# B&R Automation Studio project ComauRacer3demo
Automation Studio 4.9.2.46; technology packages: mapp 5.14.1, mappCockpit 5.14.0, mappMotion 5.14.2, mappView 5.14.2

## Configuration Racer3_demo

CPU 5APC2100.BY44-000, AutomationRuntime C4.83, Build 4.1.2, Vc V4.72.2

### Task classes (Cpu.sw)
```
Cyclic#4:
  Control <- Racer3.Control.prg
Libraries: MpRobotics, McAxGroup, MpBase, McBase, CoTrace, AsZip, FileIO, runtime, MpAlarmX, astime, MpAudit, MpRecipe, sys_lib, MpServer, MpUserX
```

### AxesGrpR3.axesgroup - 5APC2100_BY44_000/mappMotion/ComauRacer3/AxesGrpR3.axesgroup
```
Element gAxesGroup (Type=axesgroup)
  Type = PathGenAxesGroup
    ProcessingTaskClass = 1
    License = 1
    PhysicalAxes:
      JointAxes:
        JointAxis[1]:
          Name = Q1
          AxisRef = gAxisQ1
        JointAxis[2]:
          Name = Q2
          AxisRef = gAxisQ2
        JointAxis[3]:
          Name = Q3
          AxisRef = gAxisQ3
        JointAxis[4]:
          Name = Q4
          AxisRef = gAxisQ4
        JointAxis[5]:
          Name = Q5
          AxisRef = gAxisQ5
        JointAxis[6]:
          Name = Q6
          AxisRef = gAxisQ6
    MechanicalSystem:
      MechSysRef = MechSysRacer3
    BasicSettings:
      ModalDataBehaviour = ResetToDefault
      GeometryPlanning:
        TCPResolution:
          LengthResolution = 0.001
          AngleResolution = 0.001
        RoundingMode = Standard
        MaxCornerDeviation = 0.0
        MaxTangentialTransitionDeviation = 0.05
        MaxRadiusDeviation = 0.001
        WorkingPlane = XY
      TrajectoryPlanning = Basic
        LimitCheckResolution = UserDefinedTime
          Time = 0.005
        BufferTime = UserDefinedTime
          Time = 0.050
    AxesGroupFeatures:
      FeatureRef[1] = FeatureProgramsRacer3
      FeatureRef[2] = FeatureFeedForwardRacer3
      FeatureRef[3] = FeatureJoggingRacer3
  Alarms = None
```

### MotionConf.mappmotioncfg - 5APC2100_BY44_000/mappMotion/MotionConf.mappmotioncfg
```
Element MappMotionConfiguration (Type=mappmotioncfg)
```

## Configuration Racer3_working

CPU 5APC2100.BY44-000, AutomationRuntime C4.83, Build 4.1.2, Vc V4.72.2

### Task classes (Cpu.sw)
```
Cyclic#1 (cycle 2000 us, tolerance 0 us):
  Control <- Racer3.Control.prg
Cyclic#4:
  Auditing <- Auditing.prg
  Alarm <- Alarm.prg
  FileManage <- FileManager.prg
DataObjects: McAcpSys
Binaries: TCLang, McAcpDrv, McAcpSim, mvLoader, arflatprv, udbdef, TCData, mCoWebSc, McMechSys, FWRules, arcoal, arsvcreg, McPathXT, Settings, iomap, AxesR3, Role, ashwac, Hierarchy, AxGrpFtrR3, asfw, sysconf, MechSysR3, arconfig, AxesGrpR3, TC, ashwd, User, Config, Config_1, FileMngMap, Workspace, FileMngUI, ConfigF, ConfigAlmH, ConfigAdt, ConfigAlm, Config_4, Config_3, Config_2
Libraries: operator, runtime, astime, AsIecCon, MpRobotics, McAxGroup, MpBase, McBase, CoTrace, AsZip, FileIO, sys_lib, McAcpAx, McAxis, RacerLib, MpAxis, McAcpPar, McPathGen, McProgInt, MpAudit, MpServer, MpAlarmX, MpFile, AsBrStr, arssl, powerlnk, asarprof, asarlog, asio, asmem, dataobj, asepl, brsystem, aruser, MpUserX, MpFile, asbrstr, asusb
```

### Hardware
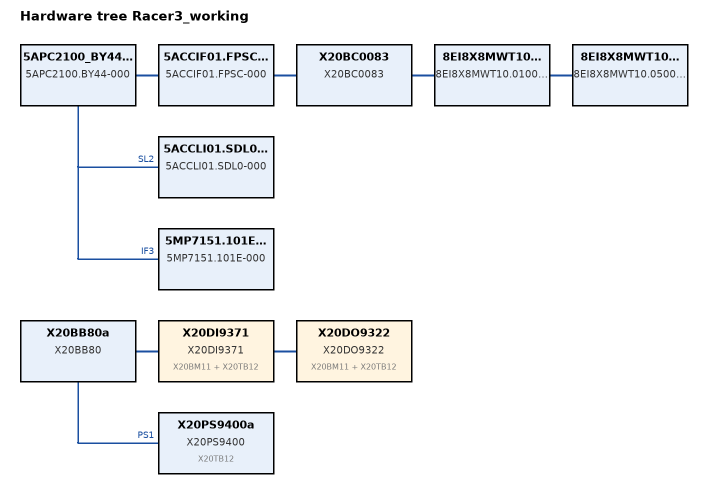
```
5ACCIF01.FPSC-000 : 5ACCIF01.FPSC-000 v1.9.0.3  [SL -> 5APC2100_BY44_000.SL1]
  Connector IF1:
    Channel1
    ChannelID1 = McAcpBroadcast
    ChannelType1 = OCTET[96]
5ACCLI01.SDL0-000 : 5ACCLI01.SDL0-000 v2.0.0.0  [SL -> 5APC2100_BY44_000.SL2]
5APC2100_BY44_000 : 5APC2100.BY44-000 v2.1.0.0
  Connector IF3:
    AssignedOperatingSystem = ARemb
    ActivateDevice = 1
    Mode = Manual
    InternetAddress = 192.168.0.100
    SubnetMask = 255.255.255.0
    ActivateSnmp = 2
  Connector IF4:
    AssignedOperatingSystem = ARemb
    ActivateDevice = 1
    Mode = Manual
    InternetAddress = 192.168.1.100
    SubnetMask = 255.255.255.0
    ActivateSnmp = 2
  Connector IF5:
    AssignedOperatingSystem = ARemb
  Connector IF6:
    AssignedOperatingSystem = ARemb
  ConfigurationID = ComauRacer3demo_czysty_racer3
  UserPartitionSize = 128
  Simulation = 1
  RemMemDevice = PCI.1.PPC21xx.SRAM
  RemMemSize = 2048
  PermanentPvSize = 768
  TimerDeviceType = EPLX2X
  TimerDevice = 5ACCIF01.FPSC-000.IF1
  TaskClassIdleTime = 2000
  Cyclic1Duration = 2000
  Cyclic1Tolerance = 0
  Cyclic1Output = 1
  FileDevice1
  FileDeviceName1 = CNC_PrgDir
  FileDevicePath1 = F:\CNC_PrgDir  // For HW config use D:\CNC_PrgDir\
  FileDevice2
  FileDeviceName2 = AUDIT
  FileDevicePath2 = F:\Audit
  FileDevice3
  FileDeviceName3 = UserPart
  FileDevicePath3 = F:\UserPart\  // For HW config use F:\
  FileDevice4
  FileDeviceName4 = RECIPE
  FileDevicePath4 = F:\Recipe
  TimeZone = 160
  ActivateDaylightSavingTime = 1
  FtpUser1
  FtpUsername1 = Admin
  FtpUserPassword1 = dPVRvIP+UG4zebJ0O0hf643aLF5yFibVmkrUfiZ9rkg=
  FtpUserSalt1 = Grtq2ClC
  FTPAccessRight1 = 0
  ActivateOpcUa = 1
  OpcUaActivateAuditEvents = 1
  OpcUa_Security_AdminRole = Everyone
  OpcUaInformationModels_PV_Version = 1
5MP7151.101E-000 : 5MP7151.101E-000 v1.1.0.0  [ETH1 -> 5APC2100_BY44_000.IF3 [Cable Type=PowerlinkCable, Length=10, Version=1.0.0.3]]
  Terminal = true
  VncKeyMappingFile = VC\5MP7151.101E-000.dis
  VncPortNumber = 5901
8EI8X8MWT10.0100-1 : 8EI8X8MWT10.0100-1 v2.3.0.3  [PLK1 -> X20BC0083.PLK2 (NodeNumber=4) [Cable Type=PowerlinkCable, Length=10, Version=1.0.0.3]; PLK2 -> 8EI8X8MWT10.0500-1.PLK1 (NodeNumber=4) [Cable Type=PowerlinkCable, Length=10, Version=1.0.0.3]]
  DriveConfiguration/Module:
    McAcoposTypeID = AcoposP3TConfig
    ActivateACOPOSSimulationOnPLC = 0
  DriveConfiguration/Encoder/EncoderX41:
    InterfaceType = EnDat
  DriveConfiguration/Encoder/EncoderX42:
    InterfaceType = EnDat
  DriveConfiguration/Encoder/EncoderX43:
    InterfaceType = EnDat
  DriveConfiguration/Channel[1]/RealAxis:
    AxisReference = gAxisQ1
  DriveConfiguration/Channel[1]/RealAxis/MechanicalElements/Gearbox:
    InputIsReadOnly = 1
    Input = 81818
    OutputIsReadOnly = 1
    Output = 1000
  DriveConfiguration/Channel[1]/RealAxis/MechanicalElements/RotaryToLinearTransformation:
    ReferenceDistanceIsReadOnly = 1
    ReferenceDistance = 360
  DriveConfiguration/Channel[1]/RealAxis/Controller:
    ModeIsReadOnly = 1
    Mode = PositionControllerWithTorqueFeedForward
  DriveConfiguration/Channel[1]/RealAxis/Controller/Mode/Position:
    ProportionalGainIsReadOnly = 1
    ProportionalGain = 75.0
    IntegrationTimeIsReadOnly = 1
    IntegrationTime = 0.0
    TotalDelayTime = 0.0004
  DriveConfiguration/Channel[1]/RealAxis/Controller/Mode/Speed:
    ProportionalGainIsReadOnly = 1
    ProportionalGain = 2.0
    IntegrationTimeIsReadOnly = 1
    IntegrationTime = 0.0
    FilterTimeIsReadOnly = 1
    FilterTime = 0.0008
  DriveConfiguration/Channel[1]/RealAxis/Controller/Mode:
    FeedForwardIsReadOnly = 1
    FeedForward = CyclicValueFromAxesGroup
  DriveConfiguration/Channel[1]/RealAxis/Controller/Mode/LoopFilters:
    LoopFilter1 = NotUsed
    LoopFilter2 = NotUsed
    LoopFilter3 = NotUsed
  DriveConfiguration/Channel[1]/RealAxis/Homing:
    Mode = RestorePosition
    RestorePositionVariable = ::gRacer3HomeRestorePos[0]
  DriveConfiguration/Channel[1]/RealAxis/StopReaction:
    Quickstop = DecelerationLimit
    DriveError = DecelerationLimit
  DriveConfiguration/Channel[1]/RealAxis/MovementErrorLimits:
    PositionError = 1.0
    VelocityErrorMonitoring = Automatic1
  DriveConfiguration/Channel[1]/RealAxis:
    JerkFilter = Used
  DriveConfiguration/Channel[1]/RealAxis/JerkFilter:
    JerkTime = 0.01
  DriveConfiguration/Channel[1]/RealAxis/DigitalInputs/HomingSwitch:
    Source = NotUsed
    Level = High
  DriveConfiguration/Channel[1]/RealAxis/DigitalInputs/PositiveLimitSwitch:
    Source = NotUsed
    Level = High
  DriveConfiguration/Channel[1]/RealAxis/DigitalInputs/NegativeLimitSwitch:
    Source = NotUsed
    Level = High
  DriveConfiguration/Channel[1]/RealAxis/DigitalInputs/Trigger1:
    Source = X8Trigger1
    Level = High
  DriveConfiguration/Channel[1]/RealAxis/DigitalInputs/Trigger2:
    Source = X8Trigger2
    Level = High
  DriveConfiguration/Channel[1]/RealAxis/DigitalInputs/Quickstop:
    Input = Trigger2
  DriveConfiguration/Channel[1]/RealAxis/Simulation:
    SimulationModeOnPLC = SetValueGeneration
    SimulationModeOnACOPOS = NotUsed
  DriveConfiguration/Channel[2]/RealAxis:
    AxisReference = gAxisQ3
  DriveConfiguration/Channel[2]/RealAxis/MechanicalElements/Gearbox:
    InputIsReadOnly = 1
    Input = 72
    OutputIsReadOnly = 1
    Output = 1
  DriveConfiguration/Channel[2]/RealAxis/MechanicalElements/RotaryToLinearTransformation:
    ReferenceDistanceIsReadOnly = 1
    ReferenceDistance = 360
  DriveConfiguration/Channel[2]/RealAxis/Controller:
    ModeIsReadOnly = 1
    Mode = PositionControllerWithTorqueFeedForward
  DriveConfiguration/Channel[2]/RealAxis/Controller/Mode/Position:
    ProportionalGainIsReadOnly = 1
    ProportionalGain = 50.0
    IntegrationTimeIsReadOnly = 1
    IntegrationTime = 0.0
    TotalDelayTime = 0.0004
  DriveConfiguration/Channel[2]/RealAxis/Controller/Mode/Speed:
    ProportionalGainIsReadOnly = 1
    ProportionalGain = 1.5
    IntegrationTimeIsReadOnly = 1
    IntegrationTime = 0.0
    FilterTimeIsReadOnly = 1
    FilterTime = 0.0008
  DriveConfiguration/Channel[2]/RealAxis/Controller/Mode:
    FeedForwardIsReadOnly = 1
    FeedForward = CyclicValueFromAxesGroup
  DriveConfiguration/Channel[2]/RealAxis/Controller/Mode/LoopFilters:
    LoopFilter1 = NotUsed
    LoopFilter2 = NotUsed
    LoopFilter3 = NotUsed
  DriveConfiguration/Channel[2]/RealAxis/Homing:
    Mode = RestorePosition
    RestorePositionVariable = ::gRacer3HomeRestorePos[2]
  DriveConfiguration/Channel[2]/RealAxis/StopReaction:
    Quickstop = DecelerationLimit
    DriveError = DecelerationLimit
  DriveConfiguration/Channel[2]/RealAxis/MovementErrorLimits:
    PositionError = 1.0
    VelocityErrorMonitoring = Automatic1
  DriveConfiguration/Channel[2]/RealAxis:
    JerkFilter = Used
  DriveConfiguration/Channel[2]/RealAxis/JerkFilter:
    JerkTime = 0.01
  DriveConfiguration/Channel[2]/RealAxis/DigitalInputs/HomingSwitch:
    Source = NotUsed
    Level = High
  DriveConfiguration/Channel[2]/RealAxis/DigitalInputs/PositiveLimitSwitch:
    Source = NotUsed
    Level = High
  DriveConfiguration/Channel[2]/RealAxis/DigitalInputs/NegativeLimitSwitch:
    Source = NotUsed
    Level = High
  DriveConfiguration/Channel[2]/RealAxis/DigitalInputs/Trigger1:
    Source = X8Trigger1
    Level = High
  DriveConfiguration/Channel[2]/RealAxis/DigitalInputs/Trigger2:
    Source = X8Trigger2
    Level = High
  DriveConfiguration/Channel[2]/RealAxis/DigitalInputs/Quickstop:
    Input = Trigger2
  DriveConfiguration/Channel[2]/RealAxis/Simulation:
    SimulationModeOnPLC = SetValueGeneration
    SimulationModeOnACOPOS = NotUsed
  DriveConfiguration/Channel[3]/RealAxis:
    AxisReference = gAxisQ5
  DriveConfiguration/Channel[3]/RealAxis/MechanicalElements/Gearbox:
    InputIsReadOnly = 1
    Input = 612
    OutputIsReadOnly = 1
    Output = 10
  DriveConfiguration/Channel[3]/RealAxis/MechanicalElements/RotaryToLinearTransformation:
    ReferenceDistanceIsReadOnly = 1
    ReferenceDistance = 360
  DriveConfiguration/Channel[3]/RealAxis/Controller:
    ModeIsReadOnly = 1
    Mode = PositionControllerWithTorqueFeedForward
  DriveConfiguration/Channel[3]/RealAxis/Controller/Mode/Position:
    ProportionalGainIsReadOnly = 1
    ProportionalGain = 200.0
    IntegrationTimeIsReadOnly = 1
    IntegrationTime = 0.0
    TotalDelayTime = 0.0004
  DriveConfiguration/Channel[3]/RealAxis/Controller/Mode/Speed:
    ProportionalGainIsReadOnly = 1
    ProportionalGain = 1.5
    IntegrationTimeIsReadOnly = 1
    IntegrationTime = 0.0
    FilterTimeIsReadOnly = 1
    FilterTime = 0.0008
  DriveConfiguration/Channel[3]/RealAxis/Controller/Mode:
    FeedForwardIsReadOnly = 1
    FeedForward = CyclicValueFromAxesGroup
  DriveConfiguration/Channel[3]/RealAxis/Controller/Mode/LoopFilters:
    LoopFilter1 = NotUsed
    LoopFilter2 = NotUsed
    LoopFilter3 = NotUsed
  DriveConfiguration/Channel[3]/RealAxis/Homing:
    Mode = RestorePosition
    RestorePositionVariable = ::gRacer3HomeRestorePos[4]
  DriveConfiguration/Channel[3]/RealAxis/StopReaction:
    Quickstop = DecelerationLimit
    DriveError = DecelerationLimit
  DriveConfiguration/Channel[3]/RealAxis/MovementErrorLimits:
    PositionError = 1.0
    VelocityErrorMonitoring = Automatic1
  DriveConfiguration/Channel[3]/RealAxis:
    JerkFilter = Used
  DriveConfiguration/Channel[3]/RealAxis/JerkFilter:
    JerkTime = 0.01
  DriveConfiguration/Channel[3]/RealAxis/DigitalInputs/HomingSwitch:
    Source = NotUsed
    Level = High
  DriveConfiguration/Channel[3]/RealAxis/DigitalInputs/PositiveLimitSwitch:
    Source = NotUsed
    Level = High
  DriveConfiguration/Channel[3]/RealAxis/DigitalInputs/NegativeLimitSwitch:
    Source = NotUsed
    Level = High
  DriveConfiguration/Channel[3]/RealAxis/DigitalInputs/Trigger1:
    Source = X8Trigger1
    Level = High
  DriveConfiguration/Channel[3]/RealAxis/DigitalInputs/Trigger2:
    Source = X8Trigger2
    Level = High
  DriveConfiguration/Channel[3]/RealAxis/DigitalInputs/Quickstop:
    Input = Trigger2
  DriveConfiguration/Channel[3]/RealAxis/Simulation:
    SimulationModeOnPLC = SetValueGeneration
    SimulationModeOnACOPOS = NotUsed
8EI8X8MWT10.0500-1 : 8EI8X8MWT10.0500-1 v2.3.0.3  [PLK1 -> 8EI8X8MWT10.0100-1.PLK2 (NodeNumber=5) [Cable Type=PowerlinkCable, Length=10, Version=1.0.0.3]]
  DriveConfiguration/Module:
    McAcoposTypeID = AcoposP3TConfig
    ActivateACOPOSSimulationOnPLC = 0
  DriveConfiguration/Encoder/EncoderX41:
    InterfaceType = EnDat
  DriveConfiguration/Encoder/EncoderX42:
    InterfaceType = EnDat
  DriveConfiguration/Encoder/EncoderX43:
    InterfaceType = EnDat
  DriveConfiguration/Channel[1]/RealAxis:
    AxisReference = gAxisQ2
  DriveConfiguration/Channel[1]/RealAxis/MechanicalElements/Gearbox:
    InputIsReadOnly = 1
    Input = 80
    OutputIsReadOnly = 1
    Output = 1
  DriveConfiguration/Channel[1]/RealAxis/MechanicalElements/RotaryToLinearTransformation:
    ReferenceDistanceIsReadOnly = 1
    ReferenceDistance = 360
  DriveConfiguration/Channel[1]/RealAxis/Controller:
    ModeIsReadOnly = 1
    Mode = PositionControllerWithTorqueFeedForward
  DriveConfiguration/Channel[1]/RealAxis/Controller/Mode/Position:
    ProportionalGainIsReadOnly = 1
    ProportionalGain = 50.0
    IntegrationTimeIsReadOnly = 1
    IntegrationTime = 0.0
    TotalDelayTime = 0.0004
  DriveConfiguration/Channel[1]/RealAxis/Controller/Mode/Speed:
    ProportionalGainIsReadOnly = 1
    ProportionalGain = 2.0
    IntegrationTimeIsReadOnly = 1
    IntegrationTime = 0.0
    FilterTimeIsReadOnly = 1
    FilterTime = 0.0008
  DriveConfiguration/Channel[1]/RealAxis/Controller/Mode:
    FeedForwardIsReadOnly = 1
    FeedForward = CyclicValueFromAxesGroup
  DriveConfiguration/Channel[1]/RealAxis/Controller/Mode/LoopFilters:
    LoopFilter1 = NotUsed
    LoopFilter2 = NotUsed
    LoopFilter3 = NotUsed
  DriveConfiguration/Channel[1]/RealAxis/Homing:
    Mode = RestorePosition
    RestorePositionVariable = ::gRacer3HomeRestorePos[1]
  DriveConfiguration/Channel[1]/RealAxis/StopReaction:
    Quickstop = DecelerationLimit
    DriveError = DecelerationLimit
  DriveConfiguration/Channel[1]/RealAxis/MovementErrorLimits:
    PositionError = 1.0
    VelocityErrorMonitoring = Automatic1
  DriveConfiguration/Channel[1]/RealAxis:
    JerkFilter = Used
  DriveConfiguration/Channel[1]/RealAxis/JerkFilter:
    JerkTime = 0.01
  DriveConfiguration/Channel[1]/RealAxis/DigitalInputs/HomingSwitch:
    Source = NotUsed
    Level = High
  DriveConfiguration/Channel[1]/RealAxis/DigitalInputs/PositiveLimitSwitch:
    Source = NotUsed
    Level = High
  DriveConfiguration/Channel[1]/RealAxis/DigitalInputs/NegativeLimitSwitch:
    Source = NotUsed
    Level = High
  DriveConfiguration/Channel[1]/RealAxis/DigitalInputs/Trigger1:
    Source = X8Trigger1
    Level = High
  DriveConfiguration/Channel[1]/RealAxis/DigitalInputs/Trigger2:
    Source = X8Trigger2
    Level = High
  DriveConfiguration/Channel[1]/RealAxis/DigitalInputs/Quickstop:
    Input = Trigger2
  DriveConfiguration/Channel[1]/RealAxis/Simulation:
    SimulationModeOnPLC = SetValueGeneration
    SimulationModeOnACOPOS = NotUsed
  DriveConfiguration/Channel[2]/RealAxis:
    AxisReference = gAxisQ4
  DriveConfiguration/Channel[2]/RealAxis/MechanicalElements/Gearbox:
    InputIsReadOnly = 1
    Input = 612
    OutputIsReadOnly = 1
    Output = 10
  DriveConfiguration/Channel[2]/RealAxis/MechanicalElements/RotaryToLinearTransformation:
    ReferenceDistanceIsReadOnly = 1
    ReferenceDistance = 360
  DriveConfiguration/Channel[2]/RealAxis/Controller:
    ModeIsReadOnly = 1
    Mode = PositionControllerWithTorqueFeedForward
  DriveConfiguration/Channel[2]/RealAxis/Controller/Mode/Position:
    ProportionalGainIsReadOnly = 1
    ProportionalGain = 100.0
    IntegrationTimeIsReadOnly = 1
    IntegrationTime = 0.0
    TotalDelayTime = 0.0004
  DriveConfiguration/Channel[2]/RealAxis/Controller/Mode/Speed:
    ProportionalGainIsReadOnly = 1
    ProportionalGain = 2.0
    IntegrationTimeIsReadOnly = 1
    IntegrationTime = 0.0
    FilterTimeIsReadOnly = 1
    FilterTime = 0.0008
  DriveConfiguration/Channel[2]/RealAxis/Controller/Mode:
    FeedForwardIsReadOnly = 1
    FeedForward = CyclicValueFromAxesGroup
  DriveConfiguration/Channel[2]/RealAxis/Controller/Mode/LoopFilters:
    LoopFilter1 = NotUsed
    LoopFilter2 = NotUsed
    LoopFilter3 = NotUsed
  DriveConfiguration/Channel[2]/RealAxis/Homing:
    Mode = RestorePosition
    RestorePositionVariable = ::gRacer3HomeRestorePos[3]
  DriveConfiguration/Channel[2]/RealAxis/StopReaction:
    Quickstop = DecelerationLimit
    DriveError = DecelerationLimit
  DriveConfiguration/Channel[2]/RealAxis/MovementErrorLimits:
    PositionError = 1.0
    VelocityErrorMonitoring = Automatic1
  DriveConfiguration/Channel[2]/RealAxis:
    JerkFilter = Used
  DriveConfiguration/Channel[2]/RealAxis/JerkFilter:
    JerkTime = 0.01
  DriveConfiguration/Channel[2]/RealAxis/DigitalInputs/HomingSwitch:
    Source = NotUsed
    Level = High
  DriveConfiguration/Channel[2]/RealAxis/DigitalInputs/PositiveLimitSwitch:
    Source = NotUsed
    Level = High
  DriveConfiguration/Channel[2]/RealAxis/DigitalInputs/NegativeLimitSwitch:
    Source = NotUsed
    Level = High
  DriveConfiguration/Channel[2]/RealAxis/DigitalInputs/Trigger1:
    Source = X8Trigger1
    Level = High
  DriveConfiguration/Channel[2]/RealAxis/DigitalInputs/Trigger2:
    Source = X8Trigger2
    Level = High
  DriveConfiguration/Channel[2]/RealAxis/DigitalInputs/Quickstop:
    Input = Trigger2
  DriveConfiguration/Channel[2]/RealAxis/Simulation:
    SimulationModeOnPLC = SetValueGeneration
    SimulationModeOnACOPOS = NotUsed
  DriveConfiguration/Channel[3]/RealAxis:
    AxisReference = gAxisQ6
  DriveConfiguration/Channel[3]/RealAxis/MechanicalElements/Gearbox:
    InputIsReadOnly = 1
    Input = 40
    OutputIsReadOnly = 1
    Output = 1
  DriveConfiguration/Channel[3]/RealAxis/MechanicalElements/RotaryToLinearTransformation:
    ReferenceDistanceIsReadOnly = 1
    ReferenceDistance = 360
  DriveConfiguration/Channel[3]/RealAxis/Controller:
    ModeIsReadOnly = 1
    Mode = PositionControllerWithTorqueFeedForward
  DriveConfiguration/Channel[3]/RealAxis/Controller/Mode/Position:
    ProportionalGainIsReadOnly = 1
    ProportionalGain = 200.0
    IntegrationTimeIsReadOnly = 1
    IntegrationTime = 0.0
    TotalDelayTime = 0.0004
  DriveConfiguration/Channel[3]/RealAxis/Controller/Mode/Speed:
    ProportionalGainIsReadOnly = 1
    ProportionalGain = 1.5
    IntegrationTimeIsReadOnly = 1
    IntegrationTime = 0.0
    FilterTimeIsReadOnly = 1
    FilterTime = 0.0008
  DriveConfiguration/Channel[3]/RealAxis/Controller/Mode:
    FeedForwardIsReadOnly = 1
    FeedForward = CyclicValueFromAxesGroup
  DriveConfiguration/Channel[3]/RealAxis/Controller/Mode/LoopFilters:
    LoopFilter1 = NotUsed
    LoopFilter2 = NotUsed
    LoopFilter3 = NotUsed
  DriveConfiguration/Channel[3]/RealAxis/Homing:
    Mode = RestorePosition
    RestorePositionVariable = ::gRacer3HomeRestorePos[5]
  DriveConfiguration/Channel[3]/RealAxis/StopReaction:
    Quickstop = DecelerationLimit
    DriveError = DecelerationLimit
  DriveConfiguration/Channel[3]/RealAxis/MovementErrorLimits:
    PositionError = 1.0
    VelocityErrorMonitoring = Automatic1
  DriveConfiguration/Channel[3]/RealAxis:
    JerkFilter = Used
  DriveConfiguration/Channel[3]/RealAxis/JerkFilter:
    JerkTime = 0.01
  DriveConfiguration/Channel[3]/RealAxis/DigitalInputs/HomingSwitch:
    Source = NotUsed
    Level = High
  DriveConfiguration/Channel[3]/RealAxis/DigitalInputs/PositiveLimitSwitch:
    Source = NotUsed
    Level = High
  DriveConfiguration/Channel[3]/RealAxis/DigitalInputs/NegativeLimitSwitch:
    Source = NotUsed
    Level = High
  DriveConfiguration/Channel[3]/RealAxis/DigitalInputs/Trigger1:
    Source = X8Trigger1
    Level = High
  DriveConfiguration/Channel[3]/RealAxis/DigitalInputs/Trigger2:
    Source = X8Trigger2
    Level = High
  DriveConfiguration/Channel[3]/RealAxis/DigitalInputs/Quickstop:
    Input = Trigger2
  DriveConfiguration/Channel[3]/RealAxis/Simulation:
    SimulationModeOnPLC = SetValueGeneration
    SimulationModeOnACOPOS = NotUsed
X20BB80a : X20BB80 v1.1.0.0
X20BC0083 : X20BC0083 v2.12.0.0  [PLK1 -> 5ACCIF01.FPSC-000.IF1 (NodeNumber=3) [Cable Type=PowerlinkCable, Length=10, Version=1.0.0.3]; PLK2 -> 8EI8X8MWT10.0100-1.PLK1 (NodeNumber=3) [Cable Type=PowerlinkCable, Length=10, Version=1.0.0.3]; SL -> X20BB80a.SL1]
X20BM11 : X20BM11 v1.0.0.1  [X2X1 -> X20BB80a.IF1]
X20BM11a : X20BM11 v1.0.0.1  [X2X1 -> X20BM11.X2X2]
X20DI9371 : X20DI9371 v1.3.0.0  [SS1 -> X20TB12c.SS; SL -> X20BM11.SL1]
X20DO9322 : X20DO9322 v1.4.0.0  [SS1 -> X20TB12d.SS; SL -> X20BM11a.SL1]
X20PS9400a : X20PS9400 v1.7.0.0  [SS1 -> X20TB12a.SS; PS -> X20BB80a.PS1]
X20TB12a : X20TB12 v1.0.0.0
X20TB12c : X20TB12 v1.0.0.0
X20TB12d : X20TB12 v1.0.0.0
```

### Cpu.per - 5APC2100_BY44_000/Cpu.per
```iecst
VAR_CONFIG
	gRacer3HomeRestorePos AT %M0; (*Permanent - stores home position, set in calibration process*)
	gIsCalibrated AT %MX432; (*Flag which tells the program whether the robot has been calibrated before*)
	gRacer3ZeroPosition AT %ML436; (*Position of axes saved after calibration*)
END_VAR
```

### AxGrpFtrR3.axesgroupfeature - 5APC2100_BY44_000/mappMotion/ComauRacer3/AxGrpFtrR3.axesgroupfeature
```
Element FeatureProgramsRacer3 (Type=axesgroupfeature)
  Type = Program
    ModalDataBehaviour = UseAxesGroupSettings
    InitialSettings:
      InterpolationTypes = LinearRapid
      PositionCoordinates = Absolute
      CircleCoordinates = Relative
      JACS_ACSProgramming = JACS
      ContourConnection = Inactive
      ProgrammingUnits = UseAxesGroupSettings
      Feedrates:
        FeedPath = Standard
        FeedCharacteristic = StandardCharacteristic
        FeedType = Feedrate
        FeedReduction = Inactive
        FeedrateValue = 0.0
        InverseFeedrateValue = 0.0
        FeedratePerRevValue = 0.0
    DefaultLanguage = BRGCode
    Location = Default
      FileDevice = CNC_PrgDir
Element FeatureFeedForwardRacer3 (Type=axesgroupfeature)
  Type = FeedForward
    Mode = ComputeAndTransmit
    RiseTime = 0.25
Element FeatureJoggingRacer3 (Type=axesgroupfeature)
  Type = Jogging
Element Feature_WorkspaceMonitoring (Type=axesgroupfeature)
  Type = WorkspaceMonitoring
    ModalDataBehaviour = UseAxesGroupSettings
    WorkspaceRef = R3WorkSpace
    SelfCollisionDetection = Enabled
    FlangeWorkspace = NotUsed
```

### AxesGrpR3.axesgroup - 5APC2100_BY44_000/mappMotion/ComauRacer3/AxesGrpR3.axesgroup
```
Element gAxesGroupRacer3 (Type=axesgroup)
  Type = PathGenAxesGroup
    ProcessingTaskClass = 1
    License = 1
    PhysicalAxes:
      JointAxes:
        JointAxis[1]:
          Name = Q1
          AxisRef = gAxisQ1
        JointAxis[2]:
          Name = Q2
          AxisRef = gAxisQ2
        JointAxis[3]:
          Name = Q3
          AxisRef = gAxisQ3
        JointAxis[4]:
          Name = Q4
          AxisRef = gAxisQ4
        JointAxis[5]:
          Name = Q5
          AxisRef = gAxisQ5
        JointAxis[6]:
          Name = Q6
          AxisRef = gAxisQ6
    MechanicalSystem:
      MechSysRef = MechSysRacer3
    BasicSettings:
      ModalDataBehaviour = ResetToDefault
      GeometryPlanning:
        TCPResolution:
          LengthResolution = 0.001
          AngleResolution = 0.001
        RoundingMode = Standard
        MaxCornerDeviation = 0.0
        MaxTangentialTransitionDeviation = 0.05
        MaxRadiusDeviation = 0.001
        WorkingPlane = XY
      TrajectoryPlanning = Basic
        LimitCheckResolution = UserDefinedTime
          Time = 0.005
        BufferTime = UserDefinedTime
          Time = 0.050
    AxesGroupFeatures:
      FeatureRef[1] = FeatureProgramsRacer3  // Programs feature
      FeatureRef[2] = FeatureFeedForwardRacer3  // Feed Forward feature
      FeatureRef[3] = FeatureJoggingRacer3  // This feature enables jogging
      FeatureRef[4] = Feature_WorkspaceMonitoring  // This feature enables workspace monitoring
      FeatureRef[5] = FeatureSharedBrakesRacer3  // This feature enables shared brake operation
  Alarms = MpAlarmX
```

### AxesR3.axis - 5APC2100_BY44_000/mappMotion/ComauRacer3/AxesR3.axis
```
Element gAxisQ1 (Type=axis)
  BaseTypeIsReadOnly = 1
  BaseType = RotaryBounded
    MeasurementUnitIsReadOnly = 1
    MeasurementUnit = 17476
    MeasurementResolutionIsReadOnly = 1
    MeasurementResolution = 0.001
    CountDirectionIsReadOnly = 1
    CountDirection = Inverse
  MovementLimitsIsReadOnly = 1
  MovementLimits = InternalForPathControlledAxis
    Position:
      LowerLimitMin = -170.0
      UpperLimitMax = 170.0
      LowerLimit = -170.0
      UpperLimit = 170.0
    VelocityIsReadOnly = 1
    Velocity:
      VelocityMax = 420.0
      Velocity = 420.0
    AccelerationIsReadOnly = 1
    Acceleration:
      AccelerationMax = 1100.0
      Acceleration = 1100.0
    DecelerationIsReadOnly = 1
    Deceleration:
      DecelerationMax = 1100.0
      Deceleration = 1100.0
    JerkIsReadOnly = 1
    Jerk = Basic
      JerkMax = 3.4E38
      Jerk = 11000.0
    TorqueIsReadOnly = 1
  Alarms = MpAlarmX
Element gAxisQ2 (Type=axis)
  BaseTypeIsReadOnly = 1
  BaseType = RotaryBounded
    MeasurementUnitIsReadOnly = 1
    MeasurementUnit = 17476
    MeasurementResolutionIsReadOnly = 1
    MeasurementResolution = 0.001
    CountDirectionIsReadOnly = 1
    CountDirection = Standard
  MovementLimitsIsReadOnly = 1
  MovementLimits = InternalForPathControlledAxis
    Position:
      LowerLimitMin = -95.0
      UpperLimitMax = 135.0
      LowerLimit = -95.0
      UpperLimit = 135.0
    VelocityIsReadOnly = 1
    Velocity:
      VelocityMax = 450.0
      Velocity = 450.0
    AccelerationIsReadOnly = 1
    Acceleration:
      AccelerationMax = 750.0
      Acceleration = 750.0
    DecelerationIsReadOnly = 1
    Deceleration:
      DecelerationMax = 750.0
      Deceleration = 750.0
    JerkIsReadOnly = 1
    Jerk = Basic
      JerkMax = 3.4E38
      Jerk = 7500.0
    TorqueIsReadOnly = 1
  Alarms = MpAlarmX
Element gAxisQ3 (Type=axis)
  BaseTypeIsReadOnly = 1
  BaseType = RotaryBounded
    MeasurementUnitIsReadOnly = 1
    MeasurementUnit = 17476
    MeasurementResolutionIsReadOnly = 1
    MeasurementResolution = 0.001
    CountDirectionIsReadOnly = 1
    CountDirection = Inverse
  MovementLimitsIsReadOnly = 1
  MovementLimits = InternalForPathControlledAxis
    Position:
      LowerLimitMin = -155.0
      UpperLimitMax = 90.0
      LowerLimit = -155.0
      UpperLimit = 90.0
    VelocityIsReadOnly = 1
    Velocity:
      VelocityMax = 480.0
      Velocity = 480.0
    AccelerationIsReadOnly = 1
    Acceleration:
      AccelerationMax = 1250.0
      Acceleration = 1250.0
    DecelerationIsReadOnly = 1
    Deceleration:
      DecelerationMax = 1250.0
      Deceleration = 1250.0
    JerkIsReadOnly = 1
    Jerk = Basic
      JerkMax = 3.4E38
      Jerk = 12500.0
    TorqueIsReadOnly = 1
  Alarms = MpAlarmX
Element gAxisQ4 (Type=axis)
  BaseTypeIsReadOnly = 1
  BaseType = RotaryBounded
    MeasurementUnitIsReadOnly = 1
    MeasurementUnit = 17476
    MeasurementResolutionIsReadOnly = 1
    MeasurementResolution = 0.001
    CountDirectionIsReadOnly = 1
    CountDirection = Standard
  MovementLimitsIsReadOnly = 1
  MovementLimits = InternalForPathControlledAxis
    Position:
      LowerLimitMin = -200.0
      UpperLimitMax = 200.0
      LowerLimit = -200.0
      UpperLimit = 200.0
    VelocityIsReadOnly = 1
    Velocity:
      VelocityMax = 600.0
      Velocity = 600.0
    AccelerationIsReadOnly = 1
    Acceleration:
      AccelerationMax = 1200.0
      Acceleration = 1200.0
    DecelerationIsReadOnly = 1
    Deceleration:
      DecelerationMax = 1200.0
      Deceleration = 1200.0
    JerkIsReadOnly = 1
    Jerk = Basic
      JerkMax = 3.4E38
      Jerk = 12000.0
    TorqueIsReadOnly = 1
  Alarms = MpAlarmX
Element gAxisQ5 (Type=axis)
  BaseTypeIsReadOnly = 1
  BaseType = RotaryBounded
    MeasurementUnitIsReadOnly = 1
    MeasurementUnit = 17476
    MeasurementResolutionIsReadOnly = 1
    MeasurementResolution = 0.001
    CountDirectionIsReadOnly = 1
    CountDirection = Standard
  MovementLimitsIsReadOnly = 1
  MovementLimits = InternalForPathControlledAxis
    Position:
      LowerLimitMin = -125.0
      UpperLimitMax = 125.0
      LowerLimit = -125.0
      UpperLimit = 125.0
    VelocityIsReadOnly = 1
    Velocity:
      VelocityMax = 600.0
      Velocity = 600.0
    AccelerationIsReadOnly = 1
    Acceleration:
      AccelerationMax = 1200.0
      Acceleration = 1200.0
    DecelerationIsReadOnly = 1
    Deceleration:
      DecelerationMax = 1200.0
      Deceleration = 1200.0
    JerkIsReadOnly = 1
    Jerk = Basic
      JerkMax = 3.4E38
      Jerk = 12000.0
    TorqueIsReadOnly = 1
  Alarms = MpAlarmX
Element gAxisQ6 (Type=axis)
  BaseTypeIsReadOnly = 1
  BaseType = RotaryBounded
    MeasurementUnitIsReadOnly = 1
    MeasurementUnit = 17476
    MeasurementResolutionIsReadOnly = 1
    MeasurementResolution = 0.001
    CountDirectionIsReadOnly = 1
    CountDirection = Standard
  MovementLimitsIsReadOnly = 1
  MovementLimits = InternalForPathControlledAxis
    Position:
      LowerLimitMin = -2700.0
      UpperLimitMax = 2700.0
      LowerLimit = -2700.0
      UpperLimit = 2700.0
    VelocityIsReadOnly = 1
    Velocity:
      VelocityMax = 875.0
      Velocity = 875.0
    AccelerationIsReadOnly = 1
    Acceleration:
      AccelerationMax = 1800.0
      Acceleration = 1800.0
    DecelerationIsReadOnly = 1
    Deceleration:
      DecelerationMax = 1800.0
      Deceleration = 1800.0
    JerkIsReadOnly = 1
    Jerk = Basic
      JerkMax = 3.4E38
      Jerk = 18000.0
    TorqueIsReadOnly = 1
  Alarms = MpAlarmX
```

### MechSysR3.mechanicalsystem - 5APC2100_BY44_000/mappMotion/ComauRacer3/MechSysR3.mechanicalsystem
```
Element MechSysRacer3 (Type=mechanicalsystem)
  Type = 6AxesRoboarm
    Subtype = 6AxesRoboarmB
      Description = Standard
        Dimensions:
          TranslationFromBaseToQ1IsReadOnly = 1
          TranslationFromBaseToQ1:
            X = 0.0
            Y = 0.0
            Z = 0.0
          TranslationFromQ1ToQ2IsReadOnly = 1
          TranslationFromQ1ToQ2:
            X = 50.0
            Y = 0.0
            Z = 365.0
          TranslationFromQ2ToQ3IsReadOnly = 1
          TranslationFromQ2ToQ3:
            X = 0.0
            Y = 0.0
            Z = 270.0
          TranslationFromQ3ToQ4IsReadOnly = 1
          TranslationFromQ3ToQ4:
            X = -50.0
            Y = 0.0
            Z = 0.0
          TranslationFromQ4ToQ5IsReadOnly = 1
          TranslationFromQ4ToQ5:
            Z = 305.94
          TranslationFromQ5ToQ6IsReadOnly = 1
          TranslationFromQ5ToQ6:
            Z = 0.0
          TranslationFromQ6ToFlange:
            X = 0.0
            Y = 0.0
            Z = 80.0
        Offsets:
          JointAxisIsReadOnly = 1
          JointAxis[1] = 0.0
          JointAxis[2] = 0.0
          JointAxis[3] = 0.0
          JointAxis[4] = 0.0
          JointAxis[5] = 0.0
          JointAxis[6] = 0.0
        CountDirections:
          JointAxisIsReadOnly = 1
          JointAxis[1] = Inverse
          JointAxis[2] = Standard
          JointAxis[3] = Inverse
          JointAxis[4] = Inverse
          JointAxis[5] = Standard
          JointAxis[6] = Inverse
      CoordinatesNames = Default
        XCoordinateName = X
        YCoordinateName = Y
        ZCoordinateName = Z
        ACoordinateName = A
        BCoordinateName = B
        CCoordinateName = C
      WireFrameModel = Standard
        Q1ToQ2 = ConnectionLine
          Distance = 5
        Q2ToQ3 = ConnectionLine
          Distance = 5
        Q3ToQ4 = ConnectionLine
          Distance = 5
        Q4ToQ5 = ConnectionLine
          Distance = 5
        Q5ToQ6 = ConnectionLine
          Distance = 5
        Q6ToFlange = ConnectionLine
          Distance = 5
        FlangeToTcp = ConnectionLine
          Distance = 5
      DynamicModel = DynParTable
        TableRef
      InternalDynamicModel = Used
        TypeIsReadOnly = 1
        Type = Comau Racer 3
        Row[1]:
          Index = 0
          Value = 4
          Unit = 
          Description = TRF_DYN11D_typ
        Row[2]:
          Index = 1
          Value = 0
          Unit = 
          Description = 
        Row[3]:
          Index = 2
          Value = 0
          Unit = 
          Description = 
        Row[4]:
          Index = 3
          Value = 0.99502
          Unit = kgm^2
          Description = m1*rc1x^2+m1*rc1y^2+Jzz1+(0.0025)*m2+m2*rc2y^2+(0.5)*Jxx2+(-0.5)*Jyy2+(0.5)*Jzz2+(0.0025)*m3+m3*rc3y^2+(0.5)*Jxx3+(-0.5)*Jyy3+(0.5)*Jzz3+(0.0025)*m4+(0.0025)*m5+(0.0025)*m6+(6694.1851)*JDrive1+(-3200)*JDrive2
        Row[5]:
          Index = 4
          Value = 0
          Unit = 
          Description = 
        Row[6]:
          Index = 5
          Value = 0
          Unit = 
          Description = 
        Row[7]:
          Index = 6
          Value = 0
          Unit = 
          Description = 
        Row[8]:
          Index = 7
          Value = -0.0079739
          Unit = kgm
          Description = m2*rc2x
        Row[9]:
          Index = 8
          Value = 0
          Unit = 
          Description = 
        Row[10]:
          Index = 9
          Value = 3.2569
          Unit = kgm
          Description = m2*rc2z+(0.27)*m3+(0.27)*m4+(0.27)*m5+(0.27)*m6
        Row[11]:
          Index = 10
          Value = -0.01529
          Unit = kgm^2
          Description = m2*rc2x*rc2y
        Row[12]:
          Index = 11
          Value = 0.018218
          Unit = kgm^2
          Description = m2*rc2y*rc2z+(0.27)*m3*rc3y
        Row[13]:
          Index = 12
          Value = -0.027
          Unit = kgm^2
          Description = m2*rc2x*rc2z
        Row[14]:
          Index = 13
          Value = 0.23153
          Unit = kgm^2
          Description = m2*rc2x^2+(-0.5)*Jxx2+(0.5)*Jyy2+(0.5)*Jzz2+(3200)*JDrive2
        Row[15]:
          Index = 14
          Value = 0
          Unit = 
          Description = 
        Row[16]:
          Index = 15
          Value = 1.1014
          Unit = kgm^2
          Description = m2*rc2z^2+(0.5)*Jxx2+(0.5)*Jyy2+(-0.5)*Jzz2+(0.0729)*m3+(0.0729)*m4+(0.0729)*m5+(0.0729)*m6+(3200)*JDrive2
        Row[17]:
          Index = 16
          Value = 0
          Unit = 
          Description = 
        Row[18]:
          Index = 17
          Value = 0
          Unit = 
          Description = 
        Row[19]:
          Index = 18
          Value = 0
          Unit = 
          Description = 
        Row[20]:
          Index = 19
          Value = 0
          Unit = 
          Description = 
        Row[21]:
          Index = 20
          Value = -0.32261
          Unit = kgm
          Description = m3*rc3x+(-0.05)*m4+(-0.05)*m5+(-0.05)*m6
        Row[22]:
          Index = 21
          Value = 0
          Unit = 
          Description = 
        Row[23]:
          Index = 22
          Value = 1.1289
          Unit = kgm
          Description = m3*rc3z+m4*rc4z+(0.30594)*m5+(0.30594)*m6
        Row[24]:
          Index = 23
          Value = -0.0059741
          Unit = kgm^2
          Description = m3*rc3x*rc3y
        Row[25]:
          Index = 24
          Value = 0.048102
          Unit = kgm^2
          Description = m3*rc3y*rc3z
        Row[26]:
          Index = 25
          Value = -0.049555
          Unit = kgm^2
          Description = m3*rc3x*rc3z+(-0.05)*m4*rc4z+(-0.015297)*m5+(-0.015297)*m6
        Row[27]:
          Index = 26
          Value = -0.026241
          Unit = kgm^2
          Description = m3*rc3x^2+(-0.5)*Jxx3+(0.5)*Jyy3+(0.5)*Jzz3+(0.0025)*m4+(0.0025)*m5+(0.0025)*m6
        Row[28]:
          Index = 27
          Value = 0
          Unit = 
          Description = 
        Row[29]:
          Index = 28
          Value = 0.21145
          Unit = kgm^2
          Description = m3*rc3z^2+(0.5)*Jxx3+(0.5)*Jyy3+(-0.5)*Jzz3+m4*rc4z^2+(0.5)*Jxx4+(0.5)*Jyy4+(-0.5)*Jzz4+(0.093599)*m5+(0.093599)*m6
        Row[30]:
          Index = 29
          Value = 0
          Unit = 
          Description = 
        Row[31]:
          Index = 30
          Value = 0
          Unit = 
          Description = 
        Row[32]:
          Index = 31
          Value = 0
          Unit = 
          Description = 
        Row[33]:
          Index = 32
          Value = 0
          Unit = 
          Description = 
        Row[34]:
          Index = 33
          Value = -0.0056373
          Unit = kgm
          Description = m4*rc4x
        Row[35]:
          Index = 34
          Value = 0.011806
          Unit = kgm
          Description = m4*rc4y+m5*rc5y
        Row[36]:
          Index = 35
          Value = 0
          Unit = 
          Description = 
        Row[37]:
          Index = 36
          Value = -0.0071612
          Unit = kgm^2
          Description = m4*rc4x*rc4y
        Row[38]:
          Index = 37
          Value = -0.00018934
          Unit = kgm^2
          Description = m4*rc4y*rc4z+(0.30594)*m5*rc5y
        Row[39]:
          Index = 38
          Value = 0.002269
          Unit = kgm^2
          Description = m4*rc4x*rc4z
        Row[40]:
          Index = 39
          Value = -0.0073563
          Unit = kgm^2
          Description = m4*rc4x^2+(-0.5)*Jxx4+(0.5)*Jyy4+(0.5)*Jzz4
        Row[41]:
          Index = 40
          Value = -0.00050442
          Unit = kgm^2
          Description = m4*rc4y^2+(0.5)*Jxx4+(-0.5)*Jyy4+(0.5)*Jzz4+m5*rc5y^2+(0.5)*Jxx5+(-0.5)*Jyy5+(0.5)*Jzz5
        Row[42]:
          Index = 41
          Value = 0
          Unit = 
          Description = 
        Row[43]:
          Index = 42
          Value = 0
          Unit = 
          Description = 
        Row[44]:
          Index = 43
          Value = 0
          Unit = 
          Description = 
        Row[45]:
          Index = 44
          Value = 0
          Unit = 
          Description = 
        Row[46]:
          Index = 45
          Value = 0
          Unit = 
          Description = 
        Row[47]:
          Index = 46
          Value = -0.0030729
          Unit = kgm
          Description = m5*rc5x
        Row[48]:
          Index = 47
          Value = 0
          Unit = 
          Description = 
        Row[49]:
          Index = 48
          Value = 0.0086628
          Unit = kgm
          Description = m5*rc5z+m6*rc6z
        Row[50]:
          Index = 49
          Value = 5.0384e-05
          Unit = kgm^2
          Description = m5*rc5x*rc5y
        Row[51]:
          Index = 50
          Value = 0.004449
          Unit = kgm^2
          Description = m5*rc5y*rc5z
        Row[52]:
          Index = 51
          Value = 0.00094987
          Unit = kgm^2
          Description = m5*rc5x*rc5z
        Row[53]:
          Index = 52
          Value = -0.0039698
          Unit = kgm^2
          Description = m5*rc5x^2+(-0.5)*Jxx5+(0.5)*Jyy5+(0.5)*Jzz5
        Row[54]:
          Index = 53
          Value = 0
          Unit = 
          Description = 
        Row[55]:
          Index = 54
          Value = -0.0023413
          Unit = kgm^2
          Description = m5*rc5z^2+(0.5)*Jxx5+(0.5)*Jyy5+(-0.5)*Jzz5+m6*rc6z^2+(0.5)*Jxx6+(0.5)*Jyy6+(-0.5)*Jzz6
        Row[56]:
          Index = 55
          Value = 0
          Unit = 
          Description = 
        Row[57]:
          Index = 56
          Value = 0
          Unit = 
          Description = 
        Row[58]:
          Index = 57
          Value = 0
          Unit = 
          Description = 
        Row[59]:
          Index = 58
          Value = 0
          Unit = 
          Description = 
        Row[60]:
          Index = 59
          Value = 0.00052765
          Unit = kgm
          Description = m6*rc6x
        Row[61]:
          Index = 60
          Value = -0.0030867
          Unit = kgm
          Description = m6*rc6y
        Row[62]:
          Index = 61
          Value = 0
          Unit = 
          Description = 
        Row[63]:
          Index = 62
          Value = 5.0962e-05
          Unit = kgm^2
          Description = m6*rc6x*rc6y
        Row[64]:
          Index = 63
          Value = -0.0015762
          Unit = kgm^2
          Description = m6*rc6y*rc6z
        Row[65]:
          Index = 64
          Value = 0.0005846
          Unit = kgm^2
          Description = m6*rc6x*rc6z
        Row[66]:
          Index = 65
          Value = 0.00067399
          Unit = kgm^2
          Description = m6*rc6x^2+(-0.5)*Jxx6+(0.5)*Jyy6+(0.5)*Jzz6
        Row[67]:
          Index = 66
          Value = 0.0013929
          Unit = kgm^2
          Description = m6*rc6y^2+(0.5)*Jxx6+(-0.5)*Jyy6+(0.5)*Jzz6
        Row[68]:
          Index = 67
          Value = 0
          Unit = 
          Description = 
        Row[69]:
          Index = 68
          Value = 0
          Unit = 
          Description = 
        Row[70]:
          Index = 69
          Value = 0
          Unit = 
          Description = 
        Row[71]:
          Index = 70
          Value = 0
          Unit = 
          Description = 
        Row[72]:
          Index = 71
          Value = 0
          Unit = 
          Description = mTool
        Row[73]:
          Index = 72
          Value = 0
          Unit = 
          Description = mTool*rcToolx
        Row[74]:
          Index = 73
          Value = 0
          Unit = 
          Description = mTool*rcTooly
        Row[75]:
          Index = 74
          Value = 0
          Unit = 
          Description = mTool*rcToolz
        Row[76]:
          Index = 75
          Value = 0
          Unit = 
          Description = mTool*rcToolx*rcTooly
        Row[77]:
          Index = 76
          Value = 0
          Unit = 
          Description = mTool*rcTooly*rcToolz
        Row[78]:
          Index = 77
          Value = 0
          Unit = 
          Description = mTool*rcToolx*rcToolz
        Row[79]:
          Index = 78
          Value = 0
          Unit = 
          Description = mTool*rcToolx^2
        Row[80]:
          Index = 79
          Value = 0
          Unit = 
          Description = mTool*rcTooly^2
        Row[81]:
          Index = 80
          Value = 0
          Unit = 
          Description = mTool*rcToolz^2
        Row[82]:
          Index = 81
          Value = 0
          Unit = 
          Description = JxxTool
        Row[83]:
          Index = 82
          Value = 0
          Unit = 
          Description = JyyTool
        Row[84]:
          Index = 83
          Value = 0
          Unit = 
          Description = JzzTool
        Row[85]:
          Index = 84
          Value = 0
          Unit = 
          Description = 
        Row[86]:
          Index = 85
          Value = 0
          Unit = 
          Description = 
        Row[87]:
          Index = 86
          Value = 9.8824e-05
          Unit = kgm^2
          Description = JDrive3
        Row[88]:
          Index = 87
          Value = 5.2689e-05
          Unit = kgm^2
          Description = JDrive4
        Row[89]:
          Index = 88
          Value = 5.129e-05
          Unit = kgm^2
          Description = JDrive5
        Row[90]:
          Index = 89
          Value = 5.2318e-05
          Unit = kgm^2
          Description = JDrive6
        Row[91]:
          Index = 90
          Value = 4.1946
          Unit = Nms
          Description = dV1
        Row[92]:
          Index = 91
          Value = 7.0888
          Unit = Nms
          Description = dV2
        Row[93]:
          Index = 92
          Value = 3.1195
          Unit = Nms
          Description = dV3
        Row[94]:
          Index = 93
          Value = 1.481
          Unit = Nms
          Description = dV4
        Row[95]:
          Index = 94
          Value = 1.1989
          Unit = Nms
          Description = dV5
        Row[96]:
          Index = 95
          Value = 0.67577
          Unit = Nms
          Description = dV6
        Row[97]:
          Index = 96
          Value = 25.5954
          Unit = Nm
          Description = dC1
        Row[98]:
          Index = 97
          Value = 14.3239
          Unit = Nm
          Description = dC2
        Row[99]:
          Index = 98
          Value = 7.6123
          Unit = Nm
          Description = dC3
        Row[100]:
          Index = 99
          Value = 7.9035
          Unit = Nm
          Description = dC4
        Row[101]:
          Index = 100
          Value = 3.5858
          Unit = Nm
          Description = dC5
        Row[102]:
          Index = 101
          Value = 5.2501
          Unit = Nm
          Description = dC6
      Couplings:
        LinearCoupling[1]:
          SourceAxisIsReadOnly = 1
          SourceAxis = 5
          SourceAxisUnitsIsReadOnly = 1
          SourceAxisUnits = 1.0
          TargetJointAxisIsReadOnly = 1
          TargetJointAxis = 6
          TargetJointAxisUnitsIsReadOnly = 1
          TargetJointAxisUnits = 0.02
      JointAxesPositionLimits:
        JointAxis[1] = ConfigureJointAxesLimits
          LowerLimitMin = -170.0
          UpperLimitMax = 170.0
          LowerLimit = -170.0
          UpperLimit = 170.0
        JointAxis[2] = ConfigureJointAxesLimits
          LowerLimitMin = -95.0
          UpperLimitMax = 135.0
          LowerLimit = -95.0
          UpperLimit = 135.0
        JointAxis[3] = ConfigureJointAxesLimits
          LowerLimitMin = -155.0
          UpperLimitMax = 90.0
          LowerLimit = -155.0
          UpperLimit = 90.0
        JointAxis[4] = ConfigureJointAxesLimits
          LowerLimitMin = -200.0
          UpperLimitMax = 200.0
          LowerLimit = -200.0
          UpperLimit = 200.0
        JointAxis[5] = ConfigureJointAxesLimits
          LowerLimitMin = -125.0
          UpperLimitMax = 125.0
          LowerLimit = -125.0
          UpperLimit = 125.0
        JointAxis[6] = ConfigureJointAxesLimits
          LowerLimitMin = -2700.0
          UpperLimitMax = 2700.0
          LowerLimit = -2700.0
          UpperLimit = 2700.0
```

### Config_1.tool - 5APC2100_BY44_000/mappMotion/Config_1.tool
```
Element RobotTool_1 (Type=tool)
  ToolType = Robot
    Translation:
      X = 0.0
      Y = 0.0
      Z = 0.0
    Orientation:
      Angle1 = 0.0
      Angle2 = 0.0
      Angle3 = 0.0
```

### AlarmXHis.mpalarmxhistory - 5APC2100_BY44_000/mappServices/AlarmXHis.mpalarmxhistory
```
Element gAlarmXHistoryLink (Type=mpalarmxhistory)
  mapp.AlarmX.History:
    Auditing = MpAudit
```

### Config.mpaudittrail - 5APC2100_BY44_000/mappServices/Config.mpaudittrail
```
Element gAuditTrailLink (Type=mpaudittrail)
  Audit:
    Events:
      [0] = 16
      [1] = 2
      [2] = 18
    TextSource:
      OutputFormat = [%[TIME=%c]] [%msg]
    Export:
      Encrypt = FALSE
  Alarms = None
```

### Config.mpfilemanager - 5APC2100_BY44_000/mappServices/Config.mpfilemanager
```
Element FileManagement (Type=mpfilemanager)
  FileManager:
    Devices:
      0:
        DeviceName = USB
        Text = USB
    Access:
      0:
        Folder = *
        Roles:
          0:
            Role = Everyone
            Rights:
              Visible = TRUE
              FolderRead = TRUE
              FileRead = TRUE
              FileEdit = TRUE
              FolderEdit = TRUE
```

### ConfigAdt.mpaudittrail - 5APC2100_BY44_000/mappServices/ConfigAdt.mpaudittrail
```
Element gAuditTrail (Type=mpaudittrail)
  Audit:
    Events:
      [0] = 16
      [1] = 2
      [2] = 18
    Export:
      Encrypt = FALSE
```

### ConfigAlm.mpalarmxcore - 5APC2100_BY44_000/mappServices/ConfigAlm.mpalarmxcore
```
Element gAlarmXCore (Type=mpalarmxcore)
  mapp.AlarmX.Core.Configuration:
    [0]:
      Name = OutOfLimits
      Message = {$AlarmTexts/OutOfLimits_Alarm_text}
```

### ConfigF.mpfilemanagerui - 5APC2100_BY44_000/mappServices/ConfigF.mpfilemanagerui
```
Element gFileManagerUI (Type=mpfilemanagerui)
  Alarms = MpAlarmX
```

### Config_1.mpalarmxcore - 5APC2100_BY44_000/mappServices/Config_1.mpalarmxcore
```
Element gAlarmXCoreLink (Type=mpalarmxcore)
  mapp.AlarmX.Core.Configuration:
    [0]:
      Name = AlarmTest
      Message = AlarmTest Message
```

### Config_3.mpuserx - 5APC2100_BY44_000/mappServices/Config_3.mpuserx
```
Element UserMgmtX (Type=mpuserx)
  ServerSettings:
    Server:
      AdditionalUserData:
        [0] = mail
        [1] = telephoneNumber
  Users:
    DefUser#1:
      id = Admin
      name = Admin Adminowski
  Groups:
    DefGroup#1:
      id = Administrators
      admin = TRUE
```

### FileMngMap.mpfilemanager - 5APC2100_BY44_000/mappServices/FileMngMap.mpfilemanager
```
Element FileManagement (Type=mpfilemanager)
  FileManager:
    USB = 1
    Devices:
      0:
        DeviceName = UserPart
        Text = UserPart
      1:
        DeviceName = CNC_PrgDir
        Text = CNC_PrgDir
      2:
        DeviceName = AUDIT
        Text = Audit
    Access:
      0:
        Folder = *
        Roles:
          0:
            Role = Everyone
            Rights:
              Visible = TRUE
              FolderRead = TRUE
              FileRead = TRUE
              FileEdit = TRUE
              FolderEdit = TRUE
          1:
            Role = Administrators
            Rights:
              Visible = TRUE
              FolderRead = TRUE
              FileRead = TRUE
              FileEdit = TRUE
              FolderEdit = TRUE
          2:
            Role = Operator
            Rights:
              Visible = TRUE
              FolderRead = TRUE
              FileRead = TRUE
              FileEdit = TRUE
              FolderEdit = TRUE
```

### RecipeMng.mprecipexml - 5APC2100_BY44_000/mappServices/RecipeMng.mprecipexml
```
Element gRecipeXmlLink (Type=mprecipexml)
```

### UserMng.mpuserx - 5APC2100_BY44_000/mappServices/UserMng.mpuserx
```
Element UserMgmtX (Type=mpuserx)
  Mgr:
    EditSameLevel = TRUE
  ServerSettings:
    Server:
      AdditionalUserData:
        [0] = mail
        [1] = telephoneNumber
  Users:
    DefUser#1:
      id = Admin
      name = Admin Adminowski
  Groups:
    DefGroup#1:
      id = Administrators
      admin = TRUE
```

## Configuration czysty_racer3

### Task classes (Cpu.sw)
```
Cyclic#4:
  Control <- Racer3.Control.prg
DataObjects: McAcpSys
Binaries: arsvcreg, udbdef, mvLoader, arflatprv, McAcpDrv, arcoal, McPathXT, McMechSys, FWRules, TCData, TCLang, mCoWebSc, McAcpSim, Settings, ashwac, User, sysconf, asfw, arconfig, ashwd, Hierarchy, iomap, Role, AxesR3, AxGrpFtrR3, MechSysR3, AxesGrpR3, Config_1, Config_4, Config_3, Config_2
Libraries: CoTrace, AsZip, runtime, FileIO, MpBase, McProgInt, McAcpAx, McBase, McPathGen, McAxis, McAxGroup, MpRobotics, arssl, astime, asieccon, powerlnk, sys_lib, asarprof, asarlog, asio, asmem, asepl, brsystem, dataobj
```

### Hardware
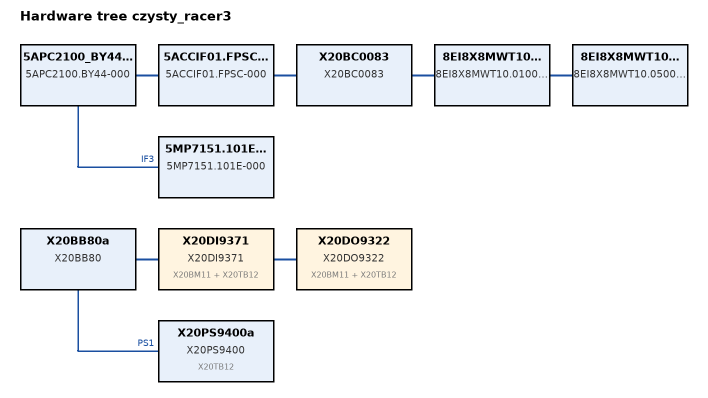
```
5ACCIF01.FPSC-000 : 5ACCIF01.FPSC-000 v1.9.0.3  [SL -> 5APC2100_BY44_000.SL1]
5APC2100_BY44_000 : 5APC2100.BY44-000 v2.1.0.0
  Connector IF3:
    AssignedOperatingSystem = ARemb
    ActivateDevice = 1
  Connector IF4:
    AssignedOperatingSystem = ARemb
    ActivateDevice = 1
  Connector IF5:
    AssignedOperatingSystem = ARemb
  Connector IF6:
    AssignedOperatingSystem = ARemb
  ConfigurationID = ComauRacer3demo_czysty_racer3
  Simulation = 1
  TimerDeviceType = EPLX2X
  TimerDevice = 5ACCIF01.FPSC-000.IF1
  TaskClassIdleTime = 2000
  FileDevice1
  FileDeviceName1 = CNC_PrgDir
  FileDevicePath1 = C:\CNC_PrgDir\
  ActivateOpcUa = 1
  OpcUaInformationModels_PV_Version = 1
5MP7151.101E-000 : 5MP7151.101E-000 v1.1.0.0  [ETH1 -> 5APC2100_BY44_000.IF3 [Cable Type=PowerlinkCable, Length=10, Version=1.0.0.3]]
  Terminal = true
  VncKeyMappingFile = VC\5MP7151.101E-000.dis
  VncPortNumber = 5901
8EI8X8MWT10.0100-1 : 8EI8X8MWT10.0100-1 v2.3.0.3  [PLK1 -> X20BC0083.PLK2 (NodeNumber=2) [Cable Type=PowerlinkCable, Length=10, Version=1.0.0.3]; PLK2 -> 8EI8X8MWT10.0500-1.PLK1 (NodeNumber=2) [Cable Type=PowerlinkCable, Length=10, Version=1.0.0.3]]
  DriveConfiguration/Module:
    McAcoposTypeID = AcoposP3TConfig
    ActivateACOPOSSimulationOnPLC = 0
  DriveConfiguration/Channel[1]/RealAxis:
    AxisReference = gAxisQ1
  DriveConfiguration/Channel[1]/RealAxis/MechanicalElements/Gearbox:
    InputIsReadOnly = 0
    Input = 1
    OutputIsReadOnly = 0
    Output = 1
  DriveConfiguration/Channel[1]/RealAxis/MechanicalElements/RotaryToLinearTransformation:
    ReferenceDistanceIsReadOnly = 0
    ReferenceDistance = 1
  DriveConfiguration/Channel[1]/RealAxis/Controller:
    ModeIsReadOnly = 0
    Mode = PositionController
  DriveConfiguration/Channel[1]/RealAxis/Controller/Mode/Position:
    ProportionalGain = 50.0
    IntegrationTime = 0.0
    PredictionTime = 0.0004
    TotalDelayTime = 0.0004
  DriveConfiguration/Channel[1]/RealAxis/Controller/Mode/Speed:
    ProportionalGainIsReadOnly = 0
    ProportionalGain = 2.0
    IntegrationTimeIsReadOnly = 0
    IntegrationTime = 0.0
    FilterTimeIsReadOnly = 0
    FilterTime = 0.0
  DriveConfiguration/Channel[1]/RealAxis/Controller/Mode/LoopFilters:
    LoopFilter1 = NotUsed
    LoopFilter2 = NotUsed
    LoopFilter3 = NotUsed
  DriveConfiguration/Channel[1]/RealAxis/Homing:
    Mode = Direct
  DriveConfiguration/Channel[1]/RealAxis/Homing/Mode:
    Position = 0.0
    ReferencePulse = NotUsed
  DriveConfiguration/Channel[1]/RealAxis/Homing:
    RestorePositionVariable = 
  DriveConfiguration/Channel[1]/RealAxis/StopReaction:
    Quickstop = DecelerationLimit
    DriveError = DecelerationLimit
  DriveConfiguration/Channel[1]/RealAxis/MovementErrorLimits:
    PositionError = 1.0
    VelocityErrorMonitoring = Automatic1
  DriveConfiguration/Channel[1]/RealAxis:
    JerkFilter = NotUsed
  DriveConfiguration/Channel[1]/RealAxis/DigitalInputs/HomingSwitch:
    Source = NotUsed
    Level = High
  DriveConfiguration/Channel[1]/RealAxis/DigitalInputs/PositiveLimitSwitch:
    Source = NotUsed
    Level = High
  DriveConfiguration/Channel[1]/RealAxis/DigitalInputs/NegativeLimitSwitch:
    Source = NotUsed
    Level = High
  DriveConfiguration/Channel[1]/RealAxis/DigitalInputs/Trigger1:
    Source = X8Trigger1
    Level = High
  DriveConfiguration/Channel[1]/RealAxis/DigitalInputs/Trigger2:
    Source = X8Trigger2
    Level = High
  DriveConfiguration/Channel[1]/RealAxis/DigitalInputs/Quickstop:
    Input = Trigger2
  DriveConfiguration/Channel[1]/RealAxis/Simulation:
    SimulationModeOnPLC = SetValueGeneration
    SimulationModeOnACOPOS = NotUsed
  DriveConfiguration/Channel[2]/RealAxis:
    AxisReference = gAxisQ2
  DriveConfiguration/Channel[2]/RealAxis/MechanicalElements/Gearbox:
    InputIsReadOnly = 0
    Input = 1
    OutputIsReadOnly = 0
    Output = 1
  DriveConfiguration/Channel[2]/RealAxis/MechanicalElements/RotaryToLinearTransformation:
    ReferenceDistanceIsReadOnly = 0
    ReferenceDistance = 1
  DriveConfiguration/Channel[2]/RealAxis/Controller:
    ModeIsReadOnly = 0
    Mode = PositionController
  DriveConfiguration/Channel[2]/RealAxis/Controller/Mode/Position:
    ProportionalGain = 50.0
    IntegrationTime = 0.0
    PredictionTime = 0.0004
    TotalDelayTime = 0.0004
  DriveConfiguration/Channel[2]/RealAxis/Controller/Mode/Speed:
    ProportionalGainIsReadOnly = 0
    ProportionalGain = 2.0
    IntegrationTimeIsReadOnly = 0
    IntegrationTime = 0.0
    FilterTimeIsReadOnly = 0
    FilterTime = 0.0
  DriveConfiguration/Channel[2]/RealAxis/Controller/Mode/LoopFilters:
    LoopFilter1 = NotUsed
    LoopFilter2 = NotUsed
    LoopFilter3 = NotUsed
  DriveConfiguration/Channel[2]/RealAxis/Homing:
    Mode = Direct
  DriveConfiguration/Channel[2]/RealAxis/Homing/Mode:
    Position = 0.0
    ReferencePulse = NotUsed
  DriveConfiguration/Channel[2]/RealAxis/Homing:
    RestorePositionVariable = 
  DriveConfiguration/Channel[2]/RealAxis/StopReaction:
    Quickstop = DecelerationLimit
    DriveError = DecelerationLimit
  DriveConfiguration/Channel[2]/RealAxis/MovementErrorLimits:
    PositionError = 1.0
    VelocityErrorMonitoring = Automatic1
  DriveConfiguration/Channel[2]/RealAxis:
    JerkFilter = NotUsed
  DriveConfiguration/Channel[2]/RealAxis/DigitalInputs/HomingSwitch:
    Source = NotUsed
    Level = High
  DriveConfiguration/Channel[2]/RealAxis/DigitalInputs/PositiveLimitSwitch:
    Source = NotUsed
    Level = High
  DriveConfiguration/Channel[2]/RealAxis/DigitalInputs/NegativeLimitSwitch:
    Source = NotUsed
    Level = High
  DriveConfiguration/Channel[2]/RealAxis/DigitalInputs/Trigger1:
    Source = X8Trigger1
    Level = High
  DriveConfiguration/Channel[2]/RealAxis/DigitalInputs/Trigger2:
    Source = X8Trigger2
    Level = High
  DriveConfiguration/Channel[2]/RealAxis/DigitalInputs/Quickstop:
    Input = Trigger2
  DriveConfiguration/Channel[2]/RealAxis/Simulation:
    SimulationModeOnPLC = SetValueGeneration
    SimulationModeOnACOPOS = NotUsed
  DriveConfiguration/Channel[3]/RealAxis:
    AxisReference = gAxisQ3
  DriveConfiguration/Channel[3]/RealAxis/MechanicalElements/Gearbox:
    InputIsReadOnly = 0
    Input = 1
    OutputIsReadOnly = 0
    Output = 1
  DriveConfiguration/Channel[3]/RealAxis/MechanicalElements/RotaryToLinearTransformation:
    ReferenceDistanceIsReadOnly = 0
    ReferenceDistance = 1
  DriveConfiguration/Channel[3]/RealAxis/Controller:
    ModeIsReadOnly = 0
    Mode = PositionController
  DriveConfiguration/Channel[3]/RealAxis/Controller/Mode/Position:
    ProportionalGain = 50.0
    IntegrationTime = 0.0
    PredictionTime = 0.0004
    TotalDelayTime = 0.0004
  DriveConfiguration/Channel[3]/RealAxis/Controller/Mode/Speed:
    ProportionalGainIsReadOnly = 0
    ProportionalGain = 2.0
    IntegrationTimeIsReadOnly = 0
    IntegrationTime = 0.0
    FilterTimeIsReadOnly = 0
    FilterTime = 0.0
  DriveConfiguration/Channel[3]/RealAxis/Controller/Mode/LoopFilters:
    LoopFilter1 = NotUsed
    LoopFilter2 = NotUsed
    LoopFilter3 = NotUsed
  DriveConfiguration/Channel[3]/RealAxis/Homing:
    Mode = Direct
  DriveConfiguration/Channel[3]/RealAxis/Homing/Mode:
    Position = 0.0
    ReferencePulse = NotUsed
  DriveConfiguration/Channel[3]/RealAxis/Homing:
    RestorePositionVariable = 
  DriveConfiguration/Channel[3]/RealAxis/StopReaction:
    Quickstop = DecelerationLimit
    DriveError = DecelerationLimit
  DriveConfiguration/Channel[3]/RealAxis/MovementErrorLimits:
    PositionError = 1.0
    VelocityErrorMonitoring = Automatic1
  DriveConfiguration/Channel[3]/RealAxis:
    JerkFilter = NotUsed
  DriveConfiguration/Channel[3]/RealAxis/DigitalInputs/HomingSwitch:
    Source = NotUsed
    Level = High
  DriveConfiguration/Channel[3]/RealAxis/DigitalInputs/PositiveLimitSwitch:
    Source = NotUsed
    Level = High
  DriveConfiguration/Channel[3]/RealAxis/DigitalInputs/NegativeLimitSwitch:
    Source = NotUsed
    Level = High
  DriveConfiguration/Channel[3]/RealAxis/DigitalInputs/Trigger1:
    Source = X8Trigger1
    Level = High
  DriveConfiguration/Channel[3]/RealAxis/DigitalInputs/Trigger2:
    Source = X8Trigger2
    Level = High
  DriveConfiguration/Channel[3]/RealAxis/DigitalInputs/Quickstop:
    Input = Trigger2
  DriveConfiguration/Channel[3]/RealAxis/Simulation:
    SimulationModeOnPLC = SetValueGeneration
    SimulationModeOnACOPOS = NotUsed
8EI8X8MWT10.0500-1 : 8EI8X8MWT10.0500-1 v2.3.0.3  [PLK1 -> 8EI8X8MWT10.0100-1.PLK2 [Cable Type=PowerlinkCable, Length=10, Version=1.0.0.3]]
  DriveConfiguration/Module:
    McAcoposTypeID = AcoposP3TConfig
    ActivateACOPOSSimulationOnPLC = 0
  DriveConfiguration/Channel[1]/RealAxis:
    AxisReference = gAxisQ4
  DriveConfiguration/Channel[1]/RealAxis/MechanicalElements/Gearbox:
    InputIsReadOnly = 0
    Input = 1
    OutputIsReadOnly = 0
    Output = 1
  DriveConfiguration/Channel[1]/RealAxis/MechanicalElements/RotaryToLinearTransformation:
    ReferenceDistanceIsReadOnly = 0
    ReferenceDistance = 1
  DriveConfiguration/Channel[1]/RealAxis/Controller:
    ModeIsReadOnly = 0
    Mode = PositionController
  DriveConfiguration/Channel[1]/RealAxis/Controller/Mode/Position:
    ProportionalGain = 50.0
    IntegrationTime = 0.0
    PredictionTime = 0.0004
    TotalDelayTime = 0.0004
  DriveConfiguration/Channel[1]/RealAxis/Controller/Mode/Speed:
    ProportionalGainIsReadOnly = 0
    ProportionalGain = 2.0
    IntegrationTimeIsReadOnly = 0
    IntegrationTime = 0.0
    FilterTimeIsReadOnly = 0
    FilterTime = 0.0
  DriveConfiguration/Channel[1]/RealAxis/Controller/Mode/LoopFilters:
    LoopFilter1 = NotUsed
    LoopFilter2 = NotUsed
    LoopFilter3 = NotUsed
  DriveConfiguration/Channel[1]/RealAxis/Homing:
    Mode = Direct
  DriveConfiguration/Channel[1]/RealAxis/Homing/Mode:
    Position = 0.0
    ReferencePulse = NotUsed
  DriveConfiguration/Channel[1]/RealAxis/Homing:
    RestorePositionVariable = 
  DriveConfiguration/Channel[1]/RealAxis/StopReaction:
    Quickstop = DecelerationLimit
    DriveError = DecelerationLimit
  DriveConfiguration/Channel[1]/RealAxis/MovementErrorLimits:
    PositionError = 1.0
    VelocityErrorMonitoring = Automatic1
  DriveConfiguration/Channel[1]/RealAxis:
    JerkFilter = NotUsed
  DriveConfiguration/Channel[1]/RealAxis/DigitalInputs/HomingSwitch:
    Source = NotUsed
    Level = High
  DriveConfiguration/Channel[1]/RealAxis/DigitalInputs/PositiveLimitSwitch:
    Source = NotUsed
    Level = High
  DriveConfiguration/Channel[1]/RealAxis/DigitalInputs/NegativeLimitSwitch:
    Source = NotUsed
    Level = High
  DriveConfiguration/Channel[1]/RealAxis/DigitalInputs/Trigger1:
    Source = X8Trigger1
    Level = High
  DriveConfiguration/Channel[1]/RealAxis/DigitalInputs/Trigger2:
    Source = X8Trigger2
    Level = High
  DriveConfiguration/Channel[1]/RealAxis/DigitalInputs/Quickstop:
    Input = Trigger2
  DriveConfiguration/Channel[1]/RealAxis/Simulation:
    SimulationModeOnPLC = SetValueGeneration
    SimulationModeOnACOPOS = NotUsed
  DriveConfiguration/Channel[2]/RealAxis:
    AxisReference = gAxisQ5
  DriveConfiguration/Channel[2]/RealAxis/MechanicalElements/Gearbox:
    InputIsReadOnly = 0
    Input = 1
    OutputIsReadOnly = 0
    Output = 1
  DriveConfiguration/Channel[2]/RealAxis/MechanicalElements/RotaryToLinearTransformation:
    ReferenceDistanceIsReadOnly = 0
    ReferenceDistance = 1
  DriveConfiguration/Channel[2]/RealAxis/Controller:
    ModeIsReadOnly = 0
    Mode = PositionController
  DriveConfiguration/Channel[2]/RealAxis/Controller/Mode/Position:
    ProportionalGain = 50.0
    IntegrationTime = 0.0
    PredictionTime = 0.0004
    TotalDelayTime = 0.0004
  DriveConfiguration/Channel[2]/RealAxis/Controller/Mode/Speed:
    ProportionalGainIsReadOnly = 0
    ProportionalGain = 2.0
    IntegrationTimeIsReadOnly = 0
    IntegrationTime = 0.0
    FilterTimeIsReadOnly = 0
    FilterTime = 0.0
  DriveConfiguration/Channel[2]/RealAxis/Controller/Mode/LoopFilters:
    LoopFilter1 = NotUsed
    LoopFilter2 = NotUsed
    LoopFilter3 = NotUsed
  DriveConfiguration/Channel[2]/RealAxis/Homing:
    Mode = Direct
  DriveConfiguration/Channel[2]/RealAxis/Homing/Mode:
    Position = 0.0
    ReferencePulse = NotUsed
  DriveConfiguration/Channel[2]/RealAxis/Homing:
    RestorePositionVariable = 
  DriveConfiguration/Channel[2]/RealAxis/StopReaction:
    Quickstop = DecelerationLimit
    DriveError = DecelerationLimit
  DriveConfiguration/Channel[2]/RealAxis/MovementErrorLimits:
    PositionError = 1.0
    VelocityErrorMonitoring = Automatic1
  DriveConfiguration/Channel[2]/RealAxis:
    JerkFilter = NotUsed
  DriveConfiguration/Channel[2]/RealAxis/DigitalInputs/HomingSwitch:
    Source = NotUsed
    Level = High
  DriveConfiguration/Channel[2]/RealAxis/DigitalInputs/PositiveLimitSwitch:
    Source = NotUsed
    Level = High
  DriveConfiguration/Channel[2]/RealAxis/DigitalInputs/NegativeLimitSwitch:
    Source = NotUsed
    Level = High
  DriveConfiguration/Channel[2]/RealAxis/DigitalInputs/Trigger1:
    Source = X8Trigger1
    Level = High
  DriveConfiguration/Channel[2]/RealAxis/DigitalInputs/Trigger2:
    Source = X8Trigger2
    Level = High
  DriveConfiguration/Channel[2]/RealAxis/DigitalInputs/Quickstop:
    Input = Trigger2
  DriveConfiguration/Channel[2]/RealAxis/Simulation:
    SimulationModeOnPLC = SetValueGeneration
    SimulationModeOnACOPOS = NotUsed
  DriveConfiguration/Channel[3]/RealAxis:
    AxisReference = gAxisQ6
  DriveConfiguration/Channel[3]/RealAxis/MechanicalElements/Gearbox:
    InputIsReadOnly = 0
    Input = 1
    OutputIsReadOnly = 0
    Output = 1
  DriveConfiguration/Channel[3]/RealAxis/MechanicalElements/RotaryToLinearTransformation:
    ReferenceDistanceIsReadOnly = 0
    ReferenceDistance = 1
  DriveConfiguration/Channel[3]/RealAxis/Controller:
    ModeIsReadOnly = 0
    Mode = PositionController
  DriveConfiguration/Channel[3]/RealAxis/Controller/Mode/Position:
    ProportionalGain = 50.0
    IntegrationTime = 0.0
    PredictionTime = 0.0004
    TotalDelayTime = 0.0004
  DriveConfiguration/Channel[3]/RealAxis/Controller/Mode/Speed:
    ProportionalGainIsReadOnly = 0
    ProportionalGain = 2.0
    IntegrationTimeIsReadOnly = 0
    IntegrationTime = 0.0
    FilterTimeIsReadOnly = 0
    FilterTime = 0.0
  DriveConfiguration/Channel[3]/RealAxis/Controller/Mode/LoopFilters:
    LoopFilter1 = NotUsed
    LoopFilter2 = NotUsed
    LoopFilter3 = NotUsed
  DriveConfiguration/Channel[3]/RealAxis/Homing:
    Mode = Direct
  DriveConfiguration/Channel[3]/RealAxis/Homing/Mode:
    Position = 0.0
    ReferencePulse = NotUsed
  DriveConfiguration/Channel[3]/RealAxis/Homing:
    RestorePositionVariable = 
  DriveConfiguration/Channel[3]/RealAxis/StopReaction:
    Quickstop = DecelerationLimit
    DriveError = DecelerationLimit
  DriveConfiguration/Channel[3]/RealAxis/MovementErrorLimits:
    PositionError = 1.0
    VelocityErrorMonitoring = Automatic1
  DriveConfiguration/Channel[3]/RealAxis:
    JerkFilter = NotUsed
  DriveConfiguration/Channel[3]/RealAxis/DigitalInputs/HomingSwitch:
    Source = NotUsed
    Level = High
  DriveConfiguration/Channel[3]/RealAxis/DigitalInputs/PositiveLimitSwitch:
    Source = NotUsed
    Level = High
  DriveConfiguration/Channel[3]/RealAxis/DigitalInputs/NegativeLimitSwitch:
    Source = NotUsed
    Level = High
  DriveConfiguration/Channel[3]/RealAxis/DigitalInputs/Trigger1:
    Source = X8Trigger1
    Level = High
  DriveConfiguration/Channel[3]/RealAxis/DigitalInputs/Trigger2:
    Source = X8Trigger2
    Level = High
  DriveConfiguration/Channel[3]/RealAxis/DigitalInputs/Quickstop:
    Input = Trigger2
  DriveConfiguration/Channel[3]/RealAxis/Simulation:
    SimulationModeOnPLC = SetValueGeneration
    SimulationModeOnACOPOS = NotUsed
X20BB80a : X20BB80 v1.1.0.0
X20BC0083 : X20BC0083 v2.12.0.0  [PLK1 -> 5ACCIF01.FPSC-000.IF1 (NodeNumber=1) [Cable Type=PowerlinkCable, Length=10, Version=1.0.0.3]; PLK2 -> 8EI8X8MWT10.0100-1.PLK1 (NodeNumber=1) [Cable Type=PowerlinkCable, Length=10, Version=1.0.0.3]; SL -> X20BB80a.SL1]
X20BM11 : X20BM11 v1.0.0.1  [X2X1 -> X20BB80a.IF1]
X20BM11a : X20BM11 v1.0.0.1  [X2X1 -> X20BM11.X2X2]
X20DI9371 : X20DI9371 v1.3.0.0  [SS1 -> X20TB12c.SS; SL -> X20BM11.SL1]
X20DO9322 : X20DO9322 v1.4.0.0  [SS1 -> X20TB12d.SS; SL -> X20BM11a.SL1]
X20PS9400a : X20PS9400 v1.7.0.0  [SS1 -> X20TB12a.SS; PS -> X20BB80a.PS1]
X20TB12a : X20TB12 v1.0.0.0
X20TB12c : X20TB12 v1.0.0.0
X20TB12d : X20TB12 v1.0.0.0
```

### Config_4.axesgroupfeature - 5APC2100_BY44_000/mappMotion/6AxesRoboArmA/Config_4.axesgroupfeature
```
Element Feature_Programs (Type=axesgroupfeature)
  Type = Program
    ModalDataBehaviour = UseAxesGroupSettings
    InitialSettings:
      InterpolationTypes = LinearRapid
      PositionCoordinates = Absolute
      CircleCoordinates = Relative
      JACS_ACSProgramming = JACS
      ContourConnection = Inactive
      ProgrammingUnits = UseAxesGroupSettings
      Feedrates:
        FeedPath = Standard
        FeedCharacteristic = StandardCharacteristic
        FeedType = Feedrate
        FeedReduction = Inactive
        FeedrateValue = 0.0
        InverseFeedrateValue = 0.0
        FeedratePerRevValue = 0.0
    DefaultLanguage = BRGCode
    Location = Default
      FileDevice = CNC_PrgDir
Element Feature_Jogging (Type=axesgroupfeature)
  Type = Jogging
```

### AxGrpFtrR3.axesgroupfeature - 5APC2100_BY44_000/mappMotion/ComauRacer3/AxGrpFtrR3.axesgroupfeature
```
Element FeatureProgramsRacer3 (Type=axesgroupfeature)
  Type = Program
    ModalDataBehaviour = UseAxesGroupSettings
    InitialSettings:
      InterpolationTypes = LinearRapid
      PositionCoordinates = Absolute
      CircleCoordinates = Relative
      JACS_ACSProgramming = JACS
      ContourConnection = Inactive
      ProgrammingUnits = UseAxesGroupSettings
      Feedrates:
        FeedPath = Standard
        FeedCharacteristic = StandardCharacteristic
        FeedType = Feedrate
        FeedReduction = Inactive
        FeedrateValue = 0.0
        InverseFeedrateValue = 0.0
        FeedratePerRevValue = 0.0
    DefaultLanguage = BRGCode
    Location = Default
      FileDevice = CNC_PrgDir
Element FeatureFeedForwardRacer3 (Type=axesgroupfeature)
  Type = FeedForward
    Mode = ComputeAndTransmit
    RiseTime = 0.25
Element FeatureJoggingRacer3 (Type=axesgroupfeature)
  Type = Jogging
```

### AxesGrpR3.axesgroup - 5APC2100_BY44_000/mappMotion/ComauRacer3/AxesGrpR3.axesgroup
```
Element gAxesGroupRacer3 (Type=axesgroup)
  Type = PathGenAxesGroup
    ProcessingTaskClass = 1
    License = 1
    PhysicalAxes:
      JointAxes:
        JointAxis[1]:
          Name = Q1
          AxisRef = gAxisQ1
        JointAxis[2]:
          Name = Q2
          AxisRef = gAxisQ2
        JointAxis[3]:
          Name = Q3
          AxisRef = gAxisQ3
        JointAxis[4]:
          Name = Q4
          AxisRef = gAxisQ4
        JointAxis[5]:
          Name = Q5
          AxisRef = gAxisQ5
        JointAxis[6]:
          Name = Q6
          AxisRef = gAxisQ6
    MechanicalSystem:
      MechSysRef = MechSysRacer3
    BasicSettings:
      ModalDataBehaviour = ResetToDefault
      GeometryPlanning:
        TCPResolution:
          LengthResolution = 0.001
          AngleResolution = 0.001
        RoundingMode = Standard
        MaxCornerDeviation = 0.0
        MaxTangentialTransitionDeviation = 0.05
        MaxRadiusDeviation = 0.001
        WorkingPlane = XY
      TrajectoryPlanning = Basic
        LimitCheckResolution = UserDefinedTime
          Time = 0.005
        BufferTime = UserDefinedTime
          Time = 0.050
    AxesGroupFeatures:
      FeatureRef[1] = FeatureProgramsRacer3
      FeatureRef[2] = FeatureFeedForwardRacer3
      FeatureRef[3] = FeatureJoggingRacer3
  Alarms = None
```

## Configuration z_helpa

CPU X20CP1586, AutomationRuntime D4.90, Build 4.1.2, Safety 0.0, Vc V4.72.2

### Task classes (Cpu.sw)
```
Cyclic#4:
  Program <- Program.prg
Libraries: McBase, MpRobotics, McAxGroup, MpBase, McPathGen, McAxis, McProgInt, McAcpAx, CoTrace, AsZip, FileIO, runtime
```

### Hardware
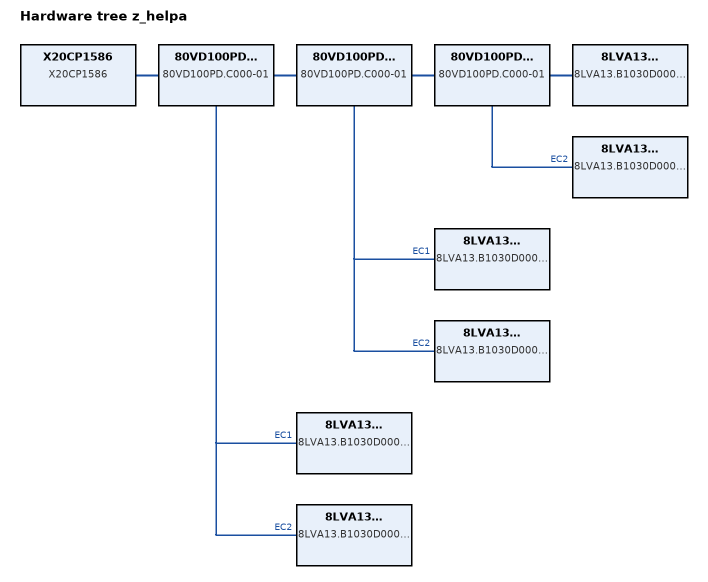
```
80VD100PD.C000-01 : 80VD100PD.C000-01 v2.5.0.0  [PLK1 -> X20CP1586.IF3 (NodeNumber=1) [Cable Type=PowerlinkCable, Length=10, Version=1.0.0.3]; PLK2 -> 80VD100PD.C000-01a.PLK1 (NodeNumber=1) [Cable Type=PowerlinkCable, Length=10, Version=1.0.0.3]; EC1 -> 8LVA13.B1030D000-0.EC; EC2 -> 8LVA13.B1030D000-0a.EC; MT2 -> 8LVA13.B1030D000-0a.MT]
  DriveConfiguration/Module:
    McAcoposTypeID = AcoposMicroDConfig
    ActivateACOPOSSimulationOnPLC = 0
  DriveConfiguration/Channel[1]/RealAxis:
    AxisReference = gAxisQ1
  DriveConfiguration/Channel[1]/RealAxis/MechanicalElements/Gearbox:
    InputIsReadOnly = 0
    Input = 1
    OutputIsReadOnly = 0
    Output = 1
  DriveConfiguration/Channel[1]/RealAxis/MechanicalElements/RotaryToLinearTransformation:
    ReferenceDistanceIsReadOnly = 0
    ReferenceDistance = 1
  DriveConfiguration/Channel[1]/RealAxis/Controller:
    ModeIsReadOnly = 0
    Mode = PositionController
  DriveConfiguration/Channel[1]/RealAxis/Controller/Mode/Position:
    ProportionalGain = 50.0
    IntegrationTime = 0.0
    PredictionTime = 0.0004
    TotalDelayTime = 0.0004
  DriveConfiguration/Channel[1]/RealAxis/Controller/Mode/Speed:
    ProportionalGainIsReadOnly = 0
    ProportionalGain = 2.0
    IntegrationTimeIsReadOnly = 0
    IntegrationTime = 0.0
    FilterTimeIsReadOnly = 0
    FilterTime = 0.0
  DriveConfiguration/Channel[1]/RealAxis/Controller/Mode/LoopFilters:
    LoopFilter1 = NotUsed
    LoopFilter2 = NotUsed
    LoopFilter3 = NotUsed
  DriveConfiguration/Channel[1]/RealAxis/Homing:
    Mode = Direct
  DriveConfiguration/Channel[1]/RealAxis/Homing/Mode:
    Position = 0.0
    ReferencePulse = NotUsed
  DriveConfiguration/Channel[1]/RealAxis/Homing:
    RestorePositionVariable = 
  DriveConfiguration/Channel[1]/RealAxis/StopReaction:
    Quickstop = DecelerationLimit
    DriveError = DecelerationLimit
  DriveConfiguration/Channel[1]/RealAxis/MovementErrorLimits:
    PositionError = 1.0
    VelocityErrorMonitoring = Automatic1
  DriveConfiguration/Channel[1]/RealAxis:
    JerkFilter = NotUsed
  DriveConfiguration/Channel[1]/RealAxis/DigitalInputs/HomingSwitch:
    Source = NotUsed
    Level = High
  DriveConfiguration/Channel[1]/RealAxis/DigitalInputs/PositiveLimitSwitch:
    Source = NotUsed
    Level = High
  DriveConfiguration/Channel[1]/RealAxis/DigitalInputs/NegativeLimitSwitch:
    Source = NotUsed
    Level = High
  DriveConfiguration/Channel[1]/RealAxis/DigitalInputs/Trigger1:
    Source = X2Trigger1
    Level = High
  DriveConfiguration/Channel[1]/RealAxis/DigitalInputs/Trigger2:
    Source = X2Trigger2
    Level = High
  DriveConfiguration/Channel[1]/RealAxis/DigitalInputs/Quickstop:
    Input = Trigger2
  DriveConfiguration/Channel[1]/RealAxis/Simulation:
    SimulationModeOnPLC = SetValueGeneration
    SimulationModeOnACOPOS = NotUsed
  DriveConfiguration/Channel[2]/RealAxis:
    AxisReference = gAxisQ2
  DriveConfiguration/Channel[2]/RealAxis/MechanicalElements/Gearbox:
    InputIsReadOnly = 0
    Input = 1
    OutputIsReadOnly = 0
    Output = 1
  DriveConfiguration/Channel[2]/RealAxis/MechanicalElements/RotaryToLinearTransformation:
    ReferenceDistanceIsReadOnly = 0
    ReferenceDistance = 1
  DriveConfiguration/Channel[2]/RealAxis/Controller:
    ModeIsReadOnly = 0
    Mode = PositionController
  DriveConfiguration/Channel[2]/RealAxis/Controller/Mode/Position:
    ProportionalGain = 50.0
    IntegrationTime = 0.0
    PredictionTime = 0.0004
    TotalDelayTime = 0.0004
  DriveConfiguration/Channel[2]/RealAxis/Controller/Mode/Speed:
    ProportionalGainIsReadOnly = 0
    ProportionalGain = 2.0
    IntegrationTimeIsReadOnly = 0
    IntegrationTime = 0.0
    FilterTimeIsReadOnly = 0
    FilterTime = 0.0
  DriveConfiguration/Channel[2]/RealAxis/Controller/Mode/LoopFilters:
    LoopFilter1 = NotUsed
    LoopFilter2 = NotUsed
    LoopFilter3 = NotUsed
  DriveConfiguration/Channel[2]/RealAxis/Homing:
    Mode = Direct
  DriveConfiguration/Channel[2]/RealAxis/Homing/Mode:
    Position = 0.0
    ReferencePulse = NotUsed
  DriveConfiguration/Channel[2]/RealAxis/Homing:
    RestorePositionVariable = 
  DriveConfiguration/Channel[2]/RealAxis/StopReaction:
    Quickstop = DecelerationLimit
    DriveError = DecelerationLimit
  DriveConfiguration/Channel[2]/RealAxis/MovementErrorLimits:
    PositionError = 1.0
    VelocityErrorMonitoring = Automatic1
  DriveConfiguration/Channel[2]/RealAxis:
    JerkFilter = NotUsed
  DriveConfiguration/Channel[2]/RealAxis/DigitalInputs/HomingSwitch:
    Source = NotUsed
    Level = High
  DriveConfiguration/Channel[2]/RealAxis/DigitalInputs/PositiveLimitSwitch:
    Source = NotUsed
    Level = High
  DriveConfiguration/Channel[2]/RealAxis/DigitalInputs/NegativeLimitSwitch:
    Source = NotUsed
    Level = High
  DriveConfiguration/Channel[2]/RealAxis/DigitalInputs/Trigger1:
    Source = X2Trigger1
    Level = High
  DriveConfiguration/Channel[2]/RealAxis/DigitalInputs/Trigger2:
    Source = X2Trigger2
    Level = High
  DriveConfiguration/Channel[2]/RealAxis/DigitalInputs/Quickstop:
    Input = Trigger2
  DriveConfiguration/Channel[2]/RealAxis/Simulation:
    SimulationModeOnPLC = SetValueGeneration
    SimulationModeOnACOPOS = NotUsed
80VD100PD.C000-01a : 80VD100PD.C000-01 v2.5.0.0  [PLK1 -> 80VD100PD.C000-01.PLK2 (NodeNumber=2) [Cable Type=PowerlinkCable, Length=10, Version=1.0.0.3]; PLK2 -> 80VD100PD.C000-01b.PLK1 (NodeNumber=2) [Cable Type=PowerlinkCable, Length=10, Version=1.0.0.3]; EC1 -> 8LVA13.B1030D000-0b.EC; EC2 -> 8LVA13.B1030D000-0c.EC; MT2 -> 8LVA13.B1030D000-0c.MT]
  DriveConfiguration/Module:
    McAcoposTypeID = AcoposMicroDConfig
    ActivateACOPOSSimulationOnPLC = 0
  DriveConfiguration/Channel[1]/RealAxis:
    AxisReference = gAxisQ3
  DriveConfiguration/Channel[1]/RealAxis/MechanicalElements/Gearbox:
    InputIsReadOnly = 0
    Input = 1
    OutputIsReadOnly = 0
    Output = 1
  DriveConfiguration/Channel[1]/RealAxis/MechanicalElements/RotaryToLinearTransformation:
    ReferenceDistanceIsReadOnly = 0
    ReferenceDistance = 1
  DriveConfiguration/Channel[1]/RealAxis/Controller:
    ModeIsReadOnly = 0
    Mode = PositionController
  DriveConfiguration/Channel[1]/RealAxis/Controller/Mode/Position:
    ProportionalGain = 50.0
    IntegrationTime = 0.0
    PredictionTime = 0.0004
    TotalDelayTime = 0.0004
  DriveConfiguration/Channel[1]/RealAxis/Controller/Mode/Speed:
    ProportionalGainIsReadOnly = 0
    ProportionalGain = 2.0
    IntegrationTimeIsReadOnly = 0
    IntegrationTime = 0.0
    FilterTimeIsReadOnly = 0
    FilterTime = 0.0
  DriveConfiguration/Channel[1]/RealAxis/Controller/Mode/LoopFilters:
    LoopFilter1 = NotUsed
    LoopFilter2 = NotUsed
    LoopFilter3 = NotUsed
  DriveConfiguration/Channel[1]/RealAxis/Homing:
    Mode = Direct
  DriveConfiguration/Channel[1]/RealAxis/Homing/Mode:
    Position = 0.0
    ReferencePulse = NotUsed
  DriveConfiguration/Channel[1]/RealAxis/Homing:
    RestorePositionVariable = 
  DriveConfiguration/Channel[1]/RealAxis/StopReaction:
    Quickstop = DecelerationLimit
    DriveError = DecelerationLimit
  DriveConfiguration/Channel[1]/RealAxis/MovementErrorLimits:
    PositionError = 1.0
    VelocityErrorMonitoring = Automatic1
  DriveConfiguration/Channel[1]/RealAxis:
    JerkFilter = NotUsed
  DriveConfiguration/Channel[1]/RealAxis/DigitalInputs/HomingSwitch:
    Source = NotUsed
    Level = High
  DriveConfiguration/Channel[1]/RealAxis/DigitalInputs/PositiveLimitSwitch:
    Source = NotUsed
    Level = High
  DriveConfiguration/Channel[1]/RealAxis/DigitalInputs/NegativeLimitSwitch:
    Source = NotUsed
    Level = High
  DriveConfiguration/Channel[1]/RealAxis/DigitalInputs/Trigger1:
    Source = X2Trigger1
    Level = High
  DriveConfiguration/Channel[1]/RealAxis/DigitalInputs/Trigger2:
    Source = X2Trigger2
    Level = High
  DriveConfiguration/Channel[1]/RealAxis/DigitalInputs/Quickstop:
    Input = Trigger2
  DriveConfiguration/Channel[1]/RealAxis/Simulation:
    SimulationModeOnPLC = SetValueGeneration
    SimulationModeOnACOPOS = NotUsed
  DriveConfiguration/Channel[2]/RealAxis:
    AxisReference = gAxisQ4
  DriveConfiguration/Channel[2]/RealAxis/MechanicalElements/Gearbox:
    InputIsReadOnly = 0
    Input = 1
    OutputIsReadOnly = 0
    Output = 1
  DriveConfiguration/Channel[2]/RealAxis/MechanicalElements/RotaryToLinearTransformation:
    ReferenceDistanceIsReadOnly = 0
    ReferenceDistance = 1
  DriveConfiguration/Channel[2]/RealAxis/Controller:
    ModeIsReadOnly = 0
    Mode = PositionController
  DriveConfiguration/Channel[2]/RealAxis/Controller/Mode/Position:
    ProportionalGain = 50.0
    IntegrationTime = 0.0
    PredictionTime = 0.0004
    TotalDelayTime = 0.0004
  DriveConfiguration/Channel[2]/RealAxis/Controller/Mode/Speed:
    ProportionalGainIsReadOnly = 0
    ProportionalGain = 2.0
    IntegrationTimeIsReadOnly = 0
    IntegrationTime = 0.0
    FilterTimeIsReadOnly = 0
    FilterTime = 0.0
  DriveConfiguration/Channel[2]/RealAxis/Controller/Mode/LoopFilters:
    LoopFilter1 = NotUsed
    LoopFilter2 = NotUsed
    LoopFilter3 = NotUsed
  DriveConfiguration/Channel[2]/RealAxis/Homing:
    Mode = Direct
  DriveConfiguration/Channel[2]/RealAxis/Homing/Mode:
    Position = 0.0
    ReferencePulse = NotUsed
  DriveConfiguration/Channel[2]/RealAxis/Homing:
    RestorePositionVariable = 
  DriveConfiguration/Channel[2]/RealAxis/StopReaction:
    Quickstop = DecelerationLimit
    DriveError = DecelerationLimit
  DriveConfiguration/Channel[2]/RealAxis/MovementErrorLimits:
    PositionError = 1.0
    VelocityErrorMonitoring = Automatic1
  DriveConfiguration/Channel[2]/RealAxis:
    JerkFilter = NotUsed
  DriveConfiguration/Channel[2]/RealAxis/DigitalInputs/HomingSwitch:
    Source = NotUsed
    Level = High
  DriveConfiguration/Channel[2]/RealAxis/DigitalInputs/PositiveLimitSwitch:
    Source = NotUsed
    Level = High
  DriveConfiguration/Channel[2]/RealAxis/DigitalInputs/NegativeLimitSwitch:
    Source = NotUsed
    Level = High
  DriveConfiguration/Channel[2]/RealAxis/DigitalInputs/Trigger1:
    Source = X2Trigger1
    Level = High
  DriveConfiguration/Channel[2]/RealAxis/DigitalInputs/Trigger2:
    Source = X2Trigger2
    Level = High
  DriveConfiguration/Channel[2]/RealAxis/DigitalInputs/Quickstop:
    Input = Trigger2
  DriveConfiguration/Channel[2]/RealAxis/Simulation:
    SimulationModeOnPLC = SetValueGeneration
    SimulationModeOnACOPOS = NotUsed
80VD100PD.C000-01b : 80VD100PD.C000-01 v2.5.0.0  [PLK1 -> 80VD100PD.C000-01a.PLK2 (NodeNumber=3) [Cable Type=PowerlinkCable, Length=10, Version=1.0.0.3]; EC1 -> 8LVA13.B1030D000-0d.EC; EC2 -> 8LVA13.B1030D000-0e.EC; MT2 -> 8LVA13.B1030D000-0e.MT]
  DriveConfiguration/Module:
    McAcoposTypeID = AcoposMicroDConfig
    ActivateACOPOSSimulationOnPLC = 0
  DriveConfiguration/Channel[1]/RealAxis:
    AxisReference = gAxisQ5
  DriveConfiguration/Channel[1]/RealAxis/MechanicalElements/Gearbox:
    InputIsReadOnly = 0
    Input = 1
    OutputIsReadOnly = 0
    Output = 1
  DriveConfiguration/Channel[1]/RealAxis/MechanicalElements/RotaryToLinearTransformation:
    ReferenceDistanceIsReadOnly = 0
    ReferenceDistance = 1
  DriveConfiguration/Channel[1]/RealAxis/Controller:
    ModeIsReadOnly = 0
    Mode = PositionController
  DriveConfiguration/Channel[1]/RealAxis/Controller/Mode/Position:
    ProportionalGain = 50.0
    IntegrationTime = 0.0
    PredictionTime = 0.0004
    TotalDelayTime = 0.0004
  DriveConfiguration/Channel[1]/RealAxis/Controller/Mode/Speed:
    ProportionalGainIsReadOnly = 0
    ProportionalGain = 2.0
    IntegrationTimeIsReadOnly = 0
    IntegrationTime = 0.0
    FilterTimeIsReadOnly = 0
    FilterTime = 0.0
  DriveConfiguration/Channel[1]/RealAxis/Controller/Mode/LoopFilters:
    LoopFilter1 = NotUsed
    LoopFilter2 = NotUsed
    LoopFilter3 = NotUsed
  DriveConfiguration/Channel[1]/RealAxis/Homing:
    Mode = Direct
  DriveConfiguration/Channel[1]/RealAxis/Homing/Mode:
    Position = 0.0
    ReferencePulse = NotUsed
  DriveConfiguration/Channel[1]/RealAxis/Homing:
    RestorePositionVariable = 
  DriveConfiguration/Channel[1]/RealAxis/StopReaction:
    Quickstop = DecelerationLimit
    DriveError = DecelerationLimit
  DriveConfiguration/Channel[1]/RealAxis/MovementErrorLimits:
    PositionError = 1.0
    VelocityErrorMonitoring = Automatic1
  DriveConfiguration/Channel[1]/RealAxis:
    JerkFilter = NotUsed
  DriveConfiguration/Channel[1]/RealAxis/DigitalInputs/HomingSwitch:
    Source = NotUsed
    Level = High
  DriveConfiguration/Channel[1]/RealAxis/DigitalInputs/PositiveLimitSwitch:
    Source = NotUsed
    Level = High
  DriveConfiguration/Channel[1]/RealAxis/DigitalInputs/NegativeLimitSwitch:
    Source = NotUsed
    Level = High
  DriveConfiguration/Channel[1]/RealAxis/DigitalInputs/Trigger1:
    Source = X2Trigger1
    Level = High
  DriveConfiguration/Channel[1]/RealAxis/DigitalInputs/Trigger2:
    Source = X2Trigger2
    Level = High
  DriveConfiguration/Channel[1]/RealAxis/DigitalInputs/Quickstop:
    Input = Trigger2
  DriveConfiguration/Channel[1]/RealAxis/Simulation:
    SimulationModeOnPLC = SetValueGeneration
    SimulationModeOnACOPOS = NotUsed
  DriveConfiguration/Channel[2]/RealAxis:
    AxisReference = gAxisQ6
  DriveConfiguration/Channel[2]/RealAxis/MechanicalElements/Gearbox:
    InputIsReadOnly = 0
    Input = 1
    OutputIsReadOnly = 0
    Output = 1
  DriveConfiguration/Channel[2]/RealAxis/MechanicalElements/RotaryToLinearTransformation:
    ReferenceDistanceIsReadOnly = 0
    ReferenceDistance = 1
  DriveConfiguration/Channel[2]/RealAxis/Controller:
    ModeIsReadOnly = 0
    Mode = PositionController
  DriveConfiguration/Channel[2]/RealAxis/Controller/Mode/Position:
    ProportionalGain = 50.0
    IntegrationTime = 0.0
    PredictionTime = 0.0004
    TotalDelayTime = 0.0004
  DriveConfiguration/Channel[2]/RealAxis/Controller/Mode/Speed:
    ProportionalGainIsReadOnly = 0
    ProportionalGain = 2.0
    IntegrationTimeIsReadOnly = 0
    IntegrationTime = 0.0
    FilterTimeIsReadOnly = 0
    FilterTime = 0.0
  DriveConfiguration/Channel[2]/RealAxis/Controller/Mode/LoopFilters:
    LoopFilter1 = NotUsed
    LoopFilter2 = NotUsed
    LoopFilter3 = NotUsed
  DriveConfiguration/Channel[2]/RealAxis/Homing:
    Mode = Direct
  DriveConfiguration/Channel[2]/RealAxis/Homing/Mode:
    Position = 0.0
    ReferencePulse = NotUsed
  DriveConfiguration/Channel[2]/RealAxis/Homing:
    RestorePositionVariable = 
  DriveConfiguration/Channel[2]/RealAxis/StopReaction:
    Quickstop = DecelerationLimit
    DriveError = DecelerationLimit
  DriveConfiguration/Channel[2]/RealAxis/MovementErrorLimits:
    PositionError = 1.0
    VelocityErrorMonitoring = Automatic1
  DriveConfiguration/Channel[2]/RealAxis:
    JerkFilter = NotUsed
  DriveConfiguration/Channel[2]/RealAxis/DigitalInputs/HomingSwitch:
    Source = NotUsed
    Level = High
  DriveConfiguration/Channel[2]/RealAxis/DigitalInputs/PositiveLimitSwitch:
    Source = NotUsed
    Level = High
  DriveConfiguration/Channel[2]/RealAxis/DigitalInputs/NegativeLimitSwitch:
    Source = NotUsed
    Level = High
  DriveConfiguration/Channel[2]/RealAxis/DigitalInputs/Trigger1:
    Source = X2Trigger1
    Level = High
  DriveConfiguration/Channel[2]/RealAxis/DigitalInputs/Trigger2:
    Source = X2Trigger2
    Level = High
  DriveConfiguration/Channel[2]/RealAxis/DigitalInputs/Quickstop:
    Input = Trigger2
  DriveConfiguration/Channel[2]/RealAxis/Simulation:
    SimulationModeOnPLC = SetValueGeneration
    SimulationModeOnACOPOS = NotUsed
8LVA13.B1030D000-0 : 8LVA13.B1030D000-0 v2.2.0.3  [EC -> 80VD100PD.C000-01.EC1; MT -> 80VD100PD.C000-01.MT1]
  M1/MotorParameters:
    MOTOR_AMB_TEMP_RATED = 40
8LVA13.B1030D000-0a : 8LVA13.B1030D000-0 v2.2.0.3  [EC -> 80VD100PD.C000-01.EC2; MT -> 80VD100PD.C000-01.MT2]
  M1/MotorParameters:
    MOTOR_AMB_TEMP_RATED = 40
8LVA13.B1030D000-0b : 8LVA13.B1030D000-0 v2.2.0.3  [EC -> 80VD100PD.C000-01a.EC1; MT -> 80VD100PD.C000-01a.MT1]
  M1/MotorParameters:
    MOTOR_AMB_TEMP_RATED = 40
8LVA13.B1030D000-0c : 8LVA13.B1030D000-0 v2.2.0.3  [EC -> 80VD100PD.C000-01a.EC2; MT -> 80VD100PD.C000-01a.MT2]
  M1/MotorParameters:
    MOTOR_AMB_TEMP_RATED = 40
8LVA13.B1030D000-0d : 8LVA13.B1030D000-0 v2.2.0.3  [EC -> 80VD100PD.C000-01b.EC1; MT -> 80VD100PD.C000-01b.MT1]
  M1/MotorParameters:
    MOTOR_AMB_TEMP_RATED = 40
8LVA13.B1030D000-0e : 8LVA13.B1030D000-0 v2.2.0.3  [EC -> 80VD100PD.C000-01b.EC2; MT -> 80VD100PD.C000-01b.MT2]
  M1/MotorParameters:
    MOTOR_AMB_TEMP_RATED = 40
X20CP1586 : X20CP1586 v1.8.1.0
  Connector IF2:
    ActivateDevice = 1
  ConfigurationID = czysta_proba_robotics_Config1
  Simulation = 1
  ActivateOpcUa = 1
  OpcUaInformationModels_PV_Version = 1
```

### Config_1.axesgroup - X20CP1586/mappMotion/6AxesRoboArmA/Config_1.axesgroup
```
Element g6AxRobA (Type=axesgroup)
  Type = PathGenAxesGroup
    ProcessingTaskClass = 1
    License = 1
    PhysicalAxes:
      JointAxes:
        JointAxis[1]:
          Name = Q1
          AxisRef = gAxisQ1
        JointAxis[2]:
          Name = Q2
          AxisRef = gAxisQ2
        JointAxis[3]:
          Name = Q3
          AxisRef = gAxisQ3
        JointAxis[4]:
          Name = Q4
          AxisRef = gAxisQ4
        JointAxis[5]:
          Name = Q5
          AxisRef = gAxisQ5
        JointAxis[6]:
          Name = Q6
          AxisRef = gAxisQ6
    MechanicalSystem:
      MechSysRef = MechSys_6AxRobA
    BasicSettings:
      ModalDataBehaviour = ResetToDefault
      GeometryPlanning:
        TCPResolution:
          LengthResolution = 0.001
          AngleResolution = 0.001
        RoundingMode = Standard
        MaxCornerDeviation = 0.0
        MaxTangentialTransitionDeviation = 0.0
        MaxRadiusDeviation = 0.001
        WorkingPlane = XY
      TrajectoryPlanning = Basic
        LimitCheckResolution = UserDefinedTime
          Time = 0.01
        BufferTime = UserDefinedTime
          Time = 0.1
    AxesGroupFeatures:
      FeatureRef[1] = Feature_Programs
      FeatureRef[2] = Feature_Jogging
  Alarms = None
```

### Config_2.axis - X20CP1586/mappMotion/6AxesRoboArmA/Config_2.axis
```
Element gAxisQ1 (Type=axis)
  BaseTypeIsReadOnly = 0
  BaseType = RotaryBounded
    MeasurementUnitIsReadOnly = 0
    MeasurementUnit = 17476
    MeasurementResolutionIsReadOnly = 0
    MeasurementResolution = 0.01
    CountDirectionIsReadOnly = 0
    CountDirection = Standard
  MovementLimitsIsReadOnly = 0
  MovementLimits = Internal
    Position:
      LowerLimitMin = -1.79769313486231E308
      UpperLimitMax = 1.79769313486231E308
      LowerLimit = -1000.0
      UpperLimit = 1000.0
    VelocityIsReadOnly = 0
    Velocity:
      VelocityMax = 3.4E38
      Velocity = 10.0
    AccelerationIsReadOnly = 0
    Acceleration:
      AccelerationMax = 3.4E38
      Acceleration = 50.0
    DecelerationIsReadOnly = 0
    Deceleration:
      DecelerationMax = 3.4E38
      Deceleration = 50.0
  Alarms = None
Element gAxisQ2 (Type=axis)
  BaseTypeIsReadOnly = 0
  BaseType = RotaryBounded
    MeasurementUnitIsReadOnly = 0
    MeasurementUnit = 17476
    MeasurementResolutionIsReadOnly = 0
    MeasurementResolution = 0.01
    CountDirectionIsReadOnly = 0
    CountDirection = Standard
  MovementLimitsIsReadOnly = 0
  MovementLimits = Internal
    Position:
      LowerLimitMin = -1.79769313486231E308
      UpperLimitMax = 1.79769313486231E308
      LowerLimit = -1000.0
      UpperLimit = 1000.0
    VelocityIsReadOnly = 0
    Velocity:
      VelocityMax = 3.4E38
      Velocity = 10.0
    AccelerationIsReadOnly = 0
    Acceleration:
      AccelerationMax = 3.4E38
      Acceleration = 50.0
    DecelerationIsReadOnly = 0
    Deceleration:
      DecelerationMax = 3.4E38
      Deceleration = 50.0
  Alarms = None
Element gAxisQ3 (Type=axis)
  BaseTypeIsReadOnly = 0
  BaseType = RotaryBounded
    MeasurementUnitIsReadOnly = 0
    MeasurementUnit = 17476
    MeasurementResolutionIsReadOnly = 0
    MeasurementResolution = 0.01
    CountDirectionIsReadOnly = 0
    CountDirection = Standard
  MovementLimitsIsReadOnly = 0
  MovementLimits = Internal
    Position:
      LowerLimitMin = -1.79769313486231E308
      UpperLimitMax = 1.79769313486231E308
      LowerLimit = -1000.0
      UpperLimit = 1000.0
    VelocityIsReadOnly = 0
    Velocity:
      VelocityMax = 3.4E38
      Velocity = 10.0
    AccelerationIsReadOnly = 0
    Acceleration:
      AccelerationMax = 3.4E38
      Acceleration = 50.0
    DecelerationIsReadOnly = 0
    Deceleration:
      DecelerationMax = 3.4E38
      Deceleration = 50.0
  Alarms = None
Element gAxisQ4 (Type=axis)
  BaseTypeIsReadOnly = 0
  BaseType = RotaryBounded
    MeasurementUnitIsReadOnly = 0
    MeasurementUnit = 17476
    MeasurementResolutionIsReadOnly = 0
    MeasurementResolution = 0.01
    CountDirectionIsReadOnly = 0
    CountDirection = Standard
  MovementLimitsIsReadOnly = 0
  MovementLimits = Internal
    Position:
      LowerLimitMin = -1.79769313486231E308
      UpperLimitMax = 1.79769313486231E308
      LowerLimit = -1000.0
      UpperLimit = 1000.0
    VelocityIsReadOnly = 0
    Velocity:
      VelocityMax = 3.4E38
      Velocity = 10.0
    AccelerationIsReadOnly = 0
    Acceleration:
      AccelerationMax = 3.4E38
      Acceleration = 50.0
    DecelerationIsReadOnly = 0
    Deceleration:
      DecelerationMax = 3.4E38
      Deceleration = 50.0
  Alarms = None
Element gAxisQ5 (Type=axis)
  BaseTypeIsReadOnly = 0
  BaseType = RotaryBounded
    MeasurementUnitIsReadOnly = 0
    MeasurementUnit = 17476
    MeasurementResolutionIsReadOnly = 0
    MeasurementResolution = 0.01
    CountDirectionIsReadOnly = 0
    CountDirection = Standard
  MovementLimitsIsReadOnly = 0
  MovementLimits = Internal
    Position:
      LowerLimitMin = -1.79769313486231E308
      UpperLimitMax = 1.79769313486231E308
      LowerLimit = -1000.0
      UpperLimit = 1000.0
    VelocityIsReadOnly = 0
    Velocity:
      VelocityMax = 3.4E38
      Velocity = 10.0
    AccelerationIsReadOnly = 0
    Acceleration:
      AccelerationMax = 3.4E38
      Acceleration = 50.0
    DecelerationIsReadOnly = 0
    Deceleration:
      DecelerationMax = 3.4E38
      Deceleration = 50.0
  Alarms = None
Element gAxisQ6 (Type=axis)
  BaseTypeIsReadOnly = 0
  BaseType = RotaryBounded
    MeasurementUnitIsReadOnly = 0
    MeasurementUnit = 17476
    MeasurementResolutionIsReadOnly = 0
    MeasurementResolution = 0.01
    CountDirectionIsReadOnly = 0
    CountDirection = Standard
  MovementLimitsIsReadOnly = 0
  MovementLimits = Internal
    Position:
      LowerLimitMin = -1.79769313486231E308
      UpperLimitMax = 1.79769313486231E308
      LowerLimit = -1000.0
      UpperLimit = 1000.0
    VelocityIsReadOnly = 0
    Velocity:
      VelocityMax = 3.4E38
      Velocity = 10.0
    AccelerationIsReadOnly = 0
    Acceleration:
      AccelerationMax = 3.4E38
      Acceleration = 50.0
    DecelerationIsReadOnly = 0
    Deceleration:
      DecelerationMax = 3.4E38
      Deceleration = 50.0
  Alarms = None
```
